LIN {X 0,Y 480.832,Z 518.896,A -85,B 0,C 180,E1 22694.82,E2 22694.82} C_VEL
LIN {X 0,Y 480.883,Z 518.889,A -85,B 0,C 180,E1 22691.393,E2 22691.393} C_VEL
LIN {X 0,Y 480.849,Z 518.879,A -85,B 0,C 180,E1 22687.888,E2 22687.888} C_VEL
LIN {X 0,Y 480.834,Z 518.897,A -85,B 0,C 180,E1 22684.413,E2 22684.413} C_VEL
LIN {X 0,Y 480.877,Z 518.875,A -85,B 0,C 180,E1 22680.953,E2 22680.953} C_VEL
LIN {X 0,Y 480.861,Z 518.895,A -85,B 0,C 180,E1 22677.498,E2 22677.498} C_VEL
LIN {X 0,Y 480.836,Z 518.893,A -85,B 0,C 180,E1 22674.032,E2 22674.032} C_VEL
LIN {X 0,Y 480.873,Z 518.893,A -85,B 0,C 180,E1 22670.546,E2 22670.546} C_VEL
LIN {X 0,Y 480.878,Z 518.894,A -85,B 0,C 180,E1 22667.023,E2 22667.023} C_VEL
LIN {X 0,Y 480.842,Z 518.893,A -85,B 0,C 180,E1 22663.573,E2 22663.573} C_VEL
LIN {X 0,Y 480.86,Z 518.889,A -85,B 0,C 180,E1 22660.017,E2 22660.017} C_VEL
LIN {X 0,Y 480.897,Z 518.897,A -85,B 0,C 180,E1 22656.47,E2 22656.47} C_VEL
LIN {X 0,Y 480.864,Z 518.888,A -85,B 0,C 180,E1 22652.859,E2 22652.859} C_VEL
LIN {X 0,Y 480.849,Z 518.893,A -85,B 0,C 180,E1 22649.373,E2 22649.373} C_VEL
LIN {X 0,Y 480.884,Z 518.892,A -85,B 0,C 180,E1 22645.841,E2 22645.841} C_VEL
LIN {X 0,Y 480.891,Z 518.896,A -85,B 0,C 180,E1 22642.19,E2 22642.19} C_VEL
LIN {X 0,Y 480.86,Z 518.9,A -85,B 0,C 180,E1 22638.642,E2 22638.642} C_VEL
LIN {X 0,Y 480.857,Z 518.892,A -85,B 0,C 180,E1 22634.986,E2 22634.986} C_VEL
LIN {X 0,Y 480.893,Z 518.896,A -85,B 0,C 180,E1 22631.387,E2 22631.387} C_VEL
LIN {X 0,Y 480.891,Z 518.896,A -85,B 0,C 180,E1 22627.806,E2 22627.806} C_VEL
LIN {X 0,Y 480.899,Z 519.178,A -85,B 0,C 180,E1 22626.666,E2 22626.666} C_VEL
LIN {X 0,Y 489.257,Z 542.949,A -85,B 0,C 180,E1 22623.815,E2 22623.815} C_VEL
LIN {X 0,Y 491.045,Z 549.01,A -85,B 0,C 180,E1 22623.147,E2 22623.147} C_VEL
LIN {X 0,Y 488.53,Z 593.414,A -85,B 0,C 180,E1 22619.418,E2 22619.418} C_VEL
LIN {X 0,Y 487.499,Z 615.888,A -85,B 0,C 180,E1 22617.597,E2 22617.597} C_VEL
LIN {X 0,Y 489.565,Z 633.074,A -85,B 0,C 180,E1 22617.228,E2 22617.228} C_VEL
LIN {X 0,Y 487.749,Z 821.161,A -85,B 0,C 180,E1 22614.405,E2 22614.405} C_VEL
LIN {X 0,Y 487.153,Z 840.046,A -85,B 0,C 180,E1 22613.909,E2 22613.909} C_VEL
LIN {X 0,Y 486.416,Z 858.284,A -85,B 0,C 180,E1 22613.213,E2 22613.213} C_VEL
LIN {X 0,Y 485.593,Z 875.737,A -85,B 0,C 180,E1 22612.327,E2 22612.327} C_VEL
LIN {X 0,Y 484.62,Z 892.847,A -85,B 0,C 180,E1 22611.228,E2 22611.228} C_VEL
LIN {X 0,Y 483.712,Z 909.068,A -85,B 0,C 180,E1 22609.941,E2 22609.941} C_VEL
LIN {X 0,Y 482.784,Z 924.925,A -85,B 0,C 180,E1 22608.411,E2 22608.411} C_VEL
LIN {X 0,Y 481.97,Z 939.095,A -85,B 0,C 180,E1 22606.76,E2 22606.76} C_VEL
LIN {X 0,Y 481.309,Z 951.749,A -85,B 0,C 180,E1 22604.989,E2 22604.989} C_VEL
LIN {X 0,Y 480.782,Z 962.938,A -85,B 0,C 180,E1 22603.102,E2 22603.102} C_VEL
LIN {X 0,Y 480.424,Z 972.395,A -85,B 0,C 180,E1 22601.161,E2 22601.161} C_VEL
LIN {X 0,Y 480.18,Z 980.439,A -85,B 0,C 180,E1 22599.106,E2 22599.106} C_VEL
LIN {X 0,Y 480.051,Z 986.651,A -85,B 0,C 180,E1 22597.06,E2 22597.06} C_VEL
LIN {X 0,Y 479.996,Z 991.41,A -85,B 0,C 180,E1 22594.9,E2 22594.9} C_VEL
LIN {X 0,Y 479.987,Z 994.401,A -85,B 0,C 180,E1 22592.747,E2 22592.747} C_VEL
LIN {X 0,Y 479.99,Z 995.698,A -85,B 0,C 180,E1 22590.598,E2 22590.598} C_VEL
LIN {X 0,Y 479.99,Z 995.327,A -85,B 0,C 180,E1 22588.45,E2 22588.45} C_VEL
LIN {X 0,Y 479.992,Z 993.281,A -85,B 0,C 180,E1 22586.299,E2 22586.299} C_VEL
LIN {X 0,Y 480.012,Z 989.511,A -85,B 0,C 180,E1 22584.144,E2 22584.144} C_VEL
LIN {X 0,Y 480.093,Z 984.297,A -85,B 0,C 180,E1 22582.102,E2 22582.102} C_VEL
LIN {X 0,Y 480.282,Z 976.985,A -85,B 0,C 180,E1 22579.964,E2 22579.964} C_VEL
LIN {X 0,Y 480.573,Z 968.08,A -85,B 0,C 180,E1 22577.921,E2 22577.921} C_VEL
LIN {X 0,Y 480.994,Z 958.057,A -85,B 0,C 180,E1 22576.049,E2 22576.049} C_VEL
LIN {X 0,Y 481.579,Z 946.227,A -85,B 0,C 180,E1 22574.221,E2 22574.221} C_VEL
LIN {X 0,Y 482.31,Z 932.666,A -85,B 0,C 180,E1 22572.479,E2 22572.479} C_VEL
LIN {X 0,Y 483.157,Z 918.064,A -85,B 0,C 180,E1 22570.918,E2 22570.918} C_VEL
LIN {X 0,Y 484.054,Z 902.156,A -85,B 0,C 180,E1 22569.509,E2 22569.509} C_VEL
LIN {X 0,Y 485.003,Z 885.243,A -85,B 0,C 180,E1 22568.285,E2 22568.285} C_VEL
LIN {X 0,Y 485.9,Z 867.99,A -85,B 0,C 180,E1 22567.284,E2 22567.284} C_VEL
LIN {X 0,Y 486.675,Z 850.244,A -85,B 0,C 180,E1 22566.483,E2 22566.483} C_VEL
LIN {X 0,Y 487.361,Z 831.618,A -85,B 0,C 180,E1 22565.872,E2 22565.872} C_VEL
LIN {X 0,Y 487.819,Z 812.718,A -85,B 0,C 180,E1 22565.472,E2 22565.472} C_VEL
LIN {X 0,Y 489.293,Z 630.035,A -85,B 0,C 180,E1 22562.747,E2 22562.747} C_VEL
LIN {X 0,Y 487.435,Z 615.346,A -85,B 0,C 180,E1 22562.393,E2 22562.393} C_VEL
LIN {X 0,Y 489.751,Z 570.848,A -85,B 0,C 180,E1 22558.701,E2 22558.701} C_VEL
LIN {X 0,Y 491.081,Z 548.213,A -85,B 0,C 180,E1 22556.751,E2 22556.751} C_VEL
LIN {X 0,Y 484.241,Z 528.175,A -85,B 0,C 180,E1 22554.341,E2 22554.341} C_VEL
LIN {X 0,Y 480.894,Z 519.106,A -85,B 0,C 180,E1 22553.106,E2 22553.106} C_VEL
LIN {X 0,Y 480.853,Z 518.898,A -85,B 0,C 180,E1 22549.556,E2 22549.556} C_VEL
LIN {X 0,Y 480.882,Z 518.9,A -85,B 0,C 180,E1 22546.006,E2 22546.006} C_VEL
LIN {X 0,Y 480.883,Z 518.896,A -85,B 0,C 180,E1 22542.436,E2 22542.436} C_VEL
LIN {X 0,Y 480.841,Z 518.893,A -85,B 0,C 180,E1 22538.959,E2 22538.959} C_VEL
LIN {X 0,Y 480.841,Z 518.896,A -85,B 0,C 180,E1 22535.315,E2 22535.315} C_VEL
LIN {X 0,Y 480.89,Z 518.889,A -85,B 0,C 180,E1 22531.878,E2 22531.878} C_VEL
LIN {X 0,Y 480.839,Z 518.896,A -85,B 0,C 180,E1 22528.436,E2 22528.436} C_VEL
LIN {X 0,Y 480.825,Z 518.897,A -85,B 0,C 180,E1 22524.838,E2 22524.838} C_VEL
LIN {X 0,Y 480.857,Z 518.901,A -85,B 0,C 180,E1 22521.339,E2 22521.339} C_VEL
LIN {X 0,Y 480.86,Z 518.894,A -85,B 0,C 180,E1 22517.784,E2 22517.784} C_VEL
LIN {X 0,Y 480.811,Z 518.889,A -85,B 0,C 180,E1 22514.315,E2 22514.315} C_VEL
LIN {X 0,Y 480.821,Z 518.897,A -85,B 0,C 180,E1 22510.787,E2 22510.787} C_VEL
LIN {X 0,Y 480.884,Z 518.899,A -85,B 0,C 180,E1 22507.286,E2 22507.286} C_VEL
LIN {X 0,Y 480.823,Z 518.892,A -85,B 0,C 180,E1 22503.815,E2 22503.815} C_VEL
LIN {X 0,Y 480.821,Z 518.891,A -85,B 0,C 180,E1 22500.238,E2 22500.238} C_VEL
LIN {X 0,Y 480.87,Z 518.896,A -85,B 0,C 180,E1 22496.781,E2 22496.781} C_VEL
LIN {X 0,Y 480.852,Z 518.898,A -85,B 0,C 180,E1 22493.313,E2 22493.313} C_VEL
LIN {X 0,Y 480.831,Z 518.894,A -85,B 0,C 180,E1 22489.819,E2 22489.819} C_VEL
LIN {X 0,Y 480.861,Z 518.89,A -85,B 0,C 180,E1 22486.288,E2 22486.288} C_VEL
LIN {X 0,Y 480.882,Z 518.891,A -85,B 0,C 180,E1 22482.827,E2 22482.827} C_VEL
LIN {X 0,Y 480.848,Z 518.897,A -85,B 0,C 180,E1 22479.299,E2 22479.299} C_VEL
LIN {X 0,Y 480.849,Z 518.892,A -85,B 0,C 180,E1 22475.596,E2 22475.596} C_VEL
LIN {X 0,Y 480.894,Z 518.897,A -85,B 0,C 180,E1 22472.073,E2 22472.073} C_VEL
LIN {X 0,Y 480.89,Z 518.895,A -85,B 0,C 180,E1 22468.47,E2 22468.47} C_VEL
LIN {X 0,Y 480.858,Z 518.902,A -85,B 0,C 180,E1 22464.977,E2 22464.977} C_VEL
LIN {X 0,Y 480.91,Z 519.174,A -85,B 0,C 180,E1 22462.637,E2 22462.637} C_VEL
LIN {X 0,Y 485.71,Z 535.44,A -85,B 0,C 180,E1 22459.884,E2 22459.884} C_VEL
LIN {X 0,Y 487.693,Z 543.443,A -85,B 0,C 180,E1 22458.614,E2 22458.614} C_VEL
LIN {X 0,Y 486.002,Z 570.518,A -85,B 0,C 180,E1 22455.042,E2 22455.042} C_VEL
LIN {X 0,Y 484.423,Z 600.385,A -85,B 0,C 180,E1 22451.173,E2 22451.173} C_VEL
LIN {X 0,Y 483.181,Z 628.631,A -85,B 0,C 180,E1 22447.575,E2 22447.575} C_VEL
LIN {X 0,Y 483.129,Z 631.811,A -85,B 0,C 180,E1 22447.207,E2 22447.207} C_VEL
LIN {X 0,Y 484.66,Z 640.368,A -85,B 0,C 180,E1 22446.962,E2 22446.962} C_VEL
LIN {X 0,Y 484.836,Z 645.811,A -85,B 0,C 180,E1 22446.867,E2 22446.867} C_VEL
LIN {X 0,Y 483.045,Z 654.53,A -85,B 0,C 180,E1 22446.817,E2 22446.817} C_VEL
LIN {X 0,Y 478.507,Z 669.749,A -85,B 0,C 180,E1 22446.799,E2 22446.799} C_VEL
LIN {X 0,Y 477.905,Z 675.336,A -85,B 0,C 180,E1 22446.738,E2 22446.738} C_VEL
LIN {X 0,Y 477.021,Z 749.526,A -85,B 0,C 180,E1 22445.515,E2 22445.515} C_VEL
LIN {X 0,Y 476.742,Z 763.894,A -85,B 0,C 180,E1 22445.07,E2 22445.07} C_VEL
LIN {X 0,Y 476.291,Z 778.064,A -85,B 0,C 180,E1 22444.41,E2 22444.41} C_VEL
LIN {X 0,Y 475.718,Z 791.572,A -85,B 0,C 180,E1 22443.552,E2 22443.552} C_VEL
LIN {X 0,Y 475.006,Z 804.939,A -85,B 0,C 180,E1 22442.426,E2 22442.426} C_VEL
LIN {X 0,Y 474.403,Z 815.997,A -85,B 0,C 180,E1 22441.225,E2 22441.225} C_VEL
LIN {X 0,Y 473.827,Z 826.024,A -85,B 0,C 180,E1 22439.855,E2 22439.855} C_VEL
LIN {X 0,Y 473.324,Z 834.493,A -85,B 0,C 180,E1 22438.374,E2 22438.374} C_VEL
LIN {X 0,Y 472.95,Z 841.657,A -85,B 0,C 180,E1 22436.759,E2 22436.759} C_VEL
LIN {X 0,Y 472.673,Z 847.643,A -85,B 0,C 180,E1 22434.891,E2 22434.891} C_VEL
LIN {X 0,Y 472.512,Z 851.491,A -85,B 0,C 180,E1 22433.042,E2 22433.042} C_VEL
LIN {X 0,Y 472.433,Z 853.501,A -85,B 0,C 180,E1 22431.214,E2 22431.214} C_VEL
LIN {X 0,Y 472.417,Z 853.747,A -85,B 0,C 180,E1 22429.273,E2 22429.273} C_VEL
LIN {X 0,Y 472.459,Z 852.063,A -85,B 0,C 180,E1 22427.358,E2 22427.358} C_VEL
LIN {X 0,Y 472.575,Z 848.779,A -85,B 0,C 180,E1 22425.584,E2 22425.584} C_VEL
LIN {X 0,Y 472.778,Z 843.721,A -85,B 0,C 180,E1 22423.824,E2 22423.824} C_VEL
LIN {X 0,Y 473.073,Z 837.213,A -85,B 0,C 180,E1 22422.199,E2 22422.199} C_VEL
LIN {X 0,Y 473.491,Z 829.444,A -85,B 0,C 180,E1 22420.707,E2 22420.707} C_VEL
LIN {X 0,Y 474.044,Z 819.355,A -85,B 0,C 180,E1 22419.207,E2 22419.207} C_VEL
LIN {X 0,Y 474.639,Z 808.412,A -85,B 0,C 180,E1 22417.929,E2 22417.929} C_VEL
LIN {X 0,Y 475.291,Z 795.658,A -85,B 0,C 180,E1 22416.763,E2 22416.763} C_VEL
LIN {X 0,Y 475.916,Z 781.501,A -85,B 0,C 180,E1 22415.786,E2 22415.786} C_VEL
LIN {X 0,Y 476.386,Z 767.869,A -85,B 0,C 180,E1 22415.092,E2 22415.092} C_VEL
LIN {X 0,Y 476.752,Z 752.577,A -85,B 0,C 180,E1 22414.558,E2 22414.558} C_VEL
LIN {X 0,Y 476.981,Z 731.635,A -85,B 0,C 180,E1 22414.162,E2 22414.162} C_VEL
LIN {X 0,Y 477.695,Z 645.512,A -85,B 0,C 180,E1 22412.808,E2 22412.808} C_VEL
LIN {X 0,Y 475.264,Z 632.071,A -85,B 0,C 180,E1 22412.47,E2 22412.47} C_VEL
LIN {X 0,Y 475.368,Z 627.356,A -85,B 0,C 180,E1 22411.927,E2 22411.927} C_VEL
LIN {X 0,Y 476.674,Z 598.333,A -85,B 0,C 180,E1 22408.196,E2 22408.196} C_VEL
LIN {X 0,Y 478.235,Z 569.754,A -85,B 0,C 180,E1 22404.48,E2 22404.48} C_VEL
LIN {X 0,Y 479.675,Z 544.41,A -85,B 0,C 180,E1 22401.126,E2 22401.126} C_VEL
LIN {X 0,Y 474.789,Z 526.621,A -85,B 0,C 180,E1 22398.308,E2 22398.308} C_VEL
LIN {X 0,Y 472.922,Z 519.987,A -85,B 0,C 180,E1 22397.174,E2 22397.174} C_VEL
LIN {X 0,Y 472.912,Z 519.892,A -85,B 0,C 180,E1 22393.716,E2 22393.716} C_VEL
LIN {X 0,Y 472.875,Z 519.888,A -85,B 0,C 180,E1 22390.208,E2 22390.208} C_VEL
LIN {X 0,Y 472.888,Z 519.86,A -85,B 0,C 180,E1 22386.71,E2 22386.71} C_VEL
LIN {X 0,Y 472.93,Z 519.89,A -85,B 0,C 180,E1 22383.15,E2 22383.15} C_VEL
LIN {X 0,Y 472.867,Z 519.859,A -85,B 0,C 180,E1 22379.786,E2 22379.786} C_VEL
LIN {X 0,Y 472.872,Z 519.89,A -85,B 0,C 180,E1 22376.069,E2 22376.069} C_VEL
LIN {X 0,Y 472.923,Z 519.88,A -85,B 0,C 180,E1 22372.645,E2 22372.645} C_VEL
LIN {X 0,Y 472.889,Z 519.891,A -85,B 0,C 180,E1 22369.196,E2 22369.196} C_VEL
LIN {X 0,Y 472.875,Z 519.888,A -85,B 0,C 180,E1 22365.586,E2 22365.586} C_VEL
LIN {X 0,Y 472.905,Z 519.876,A -85,B 0,C 180,E1 22362.085,E2 22362.085} C_VEL
LIN {X 0,Y 472.921,Z 519.886,A -85,B 0,C 180,E1 22358.587,E2 22358.587} C_VEL
LIN {X 0,Y 472.88,Z 519.881,A -85,B 0,C 180,E1 22355.092,E2 22355.092} C_VEL
LIN {X 0,Y 472.893,Z 519.887,A -85,B 0,C 180,E1 22351.483,E2 22351.483} C_VEL
LIN {X 0,Y 472.942,Z 519.879,A -85,B 0,C 180,E1 22348.129,E2 22348.129} C_VEL
LIN {X 0,Y 472.891,Z 519.876,A -85,B 0,C 180,E1 22344.616,E2 22344.616} C_VEL
LIN {X 0,Y 472.891,Z 519.887,A -85,B 0,C 180,E1 22341.066,E2 22341.066} C_VEL
LIN {X 0,Y 472.938,Z 519.865,A -85,B 0,C 180,E1 22337.556,E2 22337.556} C_VEL
LIN {X 0,Y 472.912,Z 519.886,A -85,B 0,C 180,E1 22334.072,E2 22334.072} C_VEL
LIN {X 0,Y 472.89,Z 519.879,A -85,B 0,C 180,E1 22330.477,E2 22330.477} C_VEL
LIN {X 0,Y 472.915,Z 519.88,A -85,B 0,C 180,E1 22326.922,E2 22326.922} C_VEL
LIN {X 0,Y 472.945,Z 519.883,A -85,B 0,C 180,E1 22323.394,E2 22323.394} C_VEL
LIN {X 0,Y 472.899,Z 519.866,A -85,B 0,C 180,E1 22319.879,E2 22319.879} C_VEL
LIN {X 0,Y 472.901,Z 519.887,A -85,B 0,C 180,E1 22316.242,E2 22316.242} C_VEL
LIN {X 0,Y 472.942,Z 519.866,A -85,B 0,C 180,E1 22312.713,E2 22312.713} C_VEL
LIN {X 0,Y 472.934,Z 519.887,A -85,B 0,C 180,E1 22309.155,E2 22309.155} C_VEL
LIN {X 0,Y 472.902,Z 519.877,A -85,B 0,C 180,E1 22305.678,E2 22305.678} C_VEL
LIN {X 0,Y 472.92,Z 519.885,A -85,B 0,C 180,E1 22302.053,E2 22302.053} C_VEL
LIN {X 0,Y 472.957,Z 519.874,A -85,B 0,C 180,E1 22298.417,E2 22298.417} C_VEL
LIN {X 0,Y 472.933,Z 519.885,A -85,B 0,C 180,E1 22294.798,E2 22294.798} C_VEL
LIN {X 0,Y 472.908,Z 519.887,A -85,B 0,C 180,E1 22291.319,E2 22291.319} C_VEL
LIN {X 0,Y 472.94,Z 519.883,A -85,B 0,C 180,E1 22287.808,E2 22287.808} C_VEL
LIN {X 0,Y 472.954,Z 519.88,A -85,B 0,C 180,E1 22284.155,E2 22284.155} C_VEL
LIN {X 0,Y 472.92,Z 519.882,A -85,B 0,C 180,E1 22280.634,E2 22280.634} C_VEL
LIN {X 0,Y 472.916,Z 519.886,A -85,B 0,C 180,E1 22277.011,E2 22277.011} C_VEL
LIN {X 0,Y 472.944,Z 519.884,A -85,B 0,C 180,E1 22273.397,E2 22273.397} C_VEL
LIN {X 0,Y 472.953,Z 519.884,A -85,B 0,C 180,E1 22269.832,E2 22269.832} C_VEL
LIN {X 0,Y 472.984,Z 520.157,A -85,B 0,C 180,E1 22267.197,E2 22267.197} C_VEL
LIN {X 0,Y 481.63,Z 544.659,A -85,B 0,C 180,E1 22264.19,E2 22264.19} C_VEL
LIN {X 0,Y 483.726,Z 551.404,A -85,B 0,C 180,E1 22263.424,E2 22263.424} C_VEL
LIN {X 0,Y 481.019,Z 595.587,A -85,B 0,C 180,E1 22259.65,E2 22259.65} C_VEL
LIN {X 0,Y 479.984,Z 615.915,A -85,B 0,C 180,E1 22257.965,E2 22257.965} C_VEL
LIN {X 0,Y 482.128,Z 634.091,A -85,B 0,C 180,E1 22257.565,E2 22257.565} C_VEL
LIN {X 0,Y 480.215,Z 820.44,A -85,B 0,C 180,E1 22254.735,E2 22254.735} C_VEL
LIN {X 0,Y 479.585,Z 839.412,A -85,B 0,C 180,E1 22254.231,E2 22254.231} C_VEL
LIN {X 0,Y 478.821,Z 857.057,A -85,B 0,C 180,E1 22253.551,E2 22253.551} C_VEL
LIN {X 0,Y 477.92,Z 874.81,A -85,B 0,C 180,E1 22252.64,E2 22252.64} C_VEL
LIN {X 0,Y 476.888,Z 891.93,A -85,B 0,C 180,E1 22251.525,E2 22251.525} C_VEL
LIN {X 0,Y 475.918,Z 908.149,A -85,B 0,C 180,E1 22250.218,E2 22250.218} C_VEL
LIN {X 0,Y 474.929,Z 923.994,A -85,B 0,C 180,E1 22248.663,E2 22248.663} C_VEL
LIN {X 0,Y 474.09,Z 937.665,A -85,B 0,C 180,E1 22247.047,E2 22247.047} C_VEL
LIN {X 0,Y 473.365,Z 950.783,A -85,B 0,C 180,E1 22245.184,E2 22245.184} C_VEL
LIN {X 0,Y 472.836,Z 961.624,A -85,B 0,C 180,E1 22243.326,E2 22243.326} C_VEL
LIN {X 0,Y 472.465,Z 971.123,A -85,B 0,C 180,E1 22241.351,E2 22241.351} C_VEL
LIN {X 0,Y 472.229,Z 979.203,A -85,B 0,C 180,E1 22239.261,E2 22239.261} C_VEL
LIN {X 0,Y 472.101,Z 985.44,A -85,B 0,C 180,E1 22237.179,E2 22237.179} C_VEL
LIN {X 0,Y 472.063,Z 990.218,A -85,B 0,C 180,E1 22234.983,E2 22234.983} C_VEL
LIN {X 0,Y 472.067,Z 993.22,A -85,B 0,C 180,E1 22232.794,E2 22232.794} C_VEL
LIN {X 0,Y 472.077,Z 994.52,A -85,B 0,C 180,E1 22230.608,E2 22230.608} C_VEL
LIN {X 0,Y 472.075,Z 994.144,A -85,B 0,C 180,E1 22228.424,E2 22228.424} C_VEL
LIN {X 0,Y 472.069,Z 992.083,A -85,B 0,C 180,E1 22226.237,E2 22226.237} C_VEL
LIN {X 0,Y 472.075,Z 988.291,A -85,B 0,C 180,E1 22224.045,E2 22224.045} C_VEL
LIN {X 0,Y 472.14,Z 983.045,A -85,B 0,C 180,E1 22221.968,E2 22221.968} C_VEL
LIN {X 0,Y 472.318,Z 975.94,A -85,B 0,C 180,E1 22219.855,E2 22219.855} C_VEL
LIN {X 0,Y 472.606,Z 967.105,A -85,B 0,C 180,E1 22217.789,E2 22217.789} C_VEL
LIN {X 0,Y 473.061,Z 956.667,A -85,B 0,C 180,E1 22215.811,E2 22215.811} C_VEL
LIN {X 0,Y 473.671,Z 944.769,A -85,B 0,C 180,E1 22213.95,E2 22213.95} C_VEL
LIN {X 0,Y 474.438,Z 931.388,A -85,B 0,C 180,E1 22212.21,E2 22212.21} C_VEL
LIN {X 0,Y 475.356,Z 916.422,A -85,B 0,C 180,E1 22210.593,E2 22210.593} C_VEL
LIN {X 0,Y 476.317,Z 900.378,A -85,B 0,C 180,E1 22209.161,E2 22209.161} C_VEL
LIN {X 0,Y 477.293,Z 884.216,A -85,B 0,C 180,E1 22207.981,E2 22207.981} C_VEL
LIN {X 0,Y 478.223,Z 867.38,A -85,B 0,C 180,E1 22206.988,E2 22206.988} C_VEL
LIN {X 0,Y 479.075,Z 849.388,A -85,B 0,C 180,E1 22206.163,E2 22206.163} C_VEL
LIN {X 0,Y 479.808,Z 830.665,A -85,B 0,C 180,E1 22205.541,E2 22205.541} C_VEL
LIN {X 0,Y 480.296,Z 811.558,A -85,B 0,C 180,E1 22205.135,E2 22205.135} C_VEL
LIN {X 0,Y 481.901,Z 631.165,A -85,B 0,C 180,E1 22202.404,E2 22202.404} C_VEL
LIN {X 0,Y 479.957,Z 615.552,A -85,B 0,C 180,E1 22202.022,E2 22202.022} C_VEL
LIN {X 0,Y 482.471,Z 571.77,A -85,B 0,C 180,E1 22198.313,E2 22198.313} C_VEL
LIN {X 0,Y 483.89,Z 551.303,A -85,B 0,C 180,E1 22196.521,E2 22196.521} C_VEL
LIN {X 0,Y 477.58,Z 532.578,A -85,B 0,C 180,E1 22194.22,E2 22194.22} C_VEL
LIN {X 0,Y 472.984,Z 520.089,A -85,B 0,C 180,E1 22192.493,E2 22192.493} C_VEL
LIN {X 0,Y 472.921,Z 519.884,A -85,B 0,C 180,E1 22189.006,E2 22189.006} C_VEL
LIN {X 0,Y 472.91,Z 519.89,A -85,B 0,C 180,E1 22185.424,E2 22185.424} C_VEL
LIN {X 0,Y 472.942,Z 519.881,A -85,B 0,C 180,E1 22181.918,E2 22181.918} C_VEL
LIN {X 0,Y 472.94,Z 519.878,A -85,B 0,C 180,E1 22178.349,E2 22178.349} C_VEL
LIN {X 0,Y 472.898,Z 519.885,A -85,B 0,C 180,E1 22174.811,E2 22174.811} C_VEL
LIN {X 0,Y 472.896,Z 519.888,A -85,B 0,C 180,E1 22171.107,E2 22171.107} C_VEL
LIN {X 0,Y 472.94,Z 519.878,A -85,B 0,C 180,E1 22167.66,E2 22167.66} C_VEL
LIN {X 0,Y 472.913,Z 519.881,A -85,B 0,C 180,E1 22164.082,E2 22164.082} C_VEL
LIN {X 0,Y 472.88,Z 519.889,A -85,B 0,C 180,E1 22160.677,E2 22160.677} C_VEL
LIN {X 0,Y 472.905,Z 519.891,A -85,B 0,C 180,E1 22157.147,E2 22157.147} C_VEL
LIN {X 0,Y 472.911,Z 519.877,A -85,B 0,C 180,E1 22153.697,E2 22153.697} C_VEL
LIN {X 0,Y 472.869,Z 519.885,A -85,B 0,C 180,E1 22150.231,E2 22150.231} C_VEL
LIN {X 0,Y 472.88,Z 519.89,A -85,B 0,C 180,E1 22146.556,E2 22146.556} C_VEL
LIN {X 0,Y 472.93,Z 519.886,A -85,B 0,C 180,E1 22143.03,E2 22143.03} C_VEL
LIN {X 0,Y 472.902,Z 519.878,A -85,B 0,C 180,E1 22139.515,E2 22139.515} C_VEL
LIN {X 0,Y 472.885,Z 519.886,A -85,B 0,C 180,E1 22135.999,E2 22135.999} C_VEL
LIN {X 0,Y 472.917,Z 519.887,A -85,B 0,C 180,E1 22132.468,E2 22132.468} C_VEL
LIN {X 0,Y 472.945,Z 519.886,A -85,B 0,C 180,E1 22128.908,E2 22128.908} C_VEL
LIN {X 0,Y 472.902,Z 519.883,A -85,B 0,C 180,E1 22125.427,E2 22125.427} C_VEL
LIN {X 0,Y 472.905,Z 519.885,A -85,B 0,C 180,E1 22121.765,E2 22121.765} C_VEL
LIN {X 0,Y 472.954,Z 519.882,A -85,B 0,C 180,E1 22118.286,E2 22118.286} C_VEL
LIN {X 0,Y 472.94,Z 519.885,A -85,B 0,C 180,E1 22114.719,E2 22114.719} C_VEL
LIN {X 0,Y 472.914,Z 519.89,A -85,B 0,C 180,E1 22111.18,E2 22111.18} C_VEL
LIN {X 0,Y 472.924,Z 519.887,A -85,B 0,C 180,E1 22107.508,E2 22107.508} C_VEL
LIN {X 0,Y 472.953,Z 519.882,A -85,B 0,C 180,E1 22104.005,E2 22104.005} C_VEL
LIN {X 0,Y 472.97,Z 520.223,A -85,B 0,C 180,E1 22103.203,E2 22103.203} C_VEL
LIN {X 0,Y 477.948,Z 536.611,A -85,B 0,C 180,E1 22100.353,E2 22100.353} C_VEL
LIN {X 0,Y 480.275,Z 546.322,A -85,B 0,C 180,E1 22098.783,E2 22098.783} C_VEL
LIN {X 0,Y 478.464,Z 573.198,A -85,B 0,C 180,E1 22095.184,E2 22095.184} C_VEL
LIN {X 0,Y 476.803,Z 602.516,A -85,B 0,C 180,E1 22091.336,E2 22091.336} C_VEL
LIN {X 0,Y 475.472,Z 631.275,A -85,B 0,C 180,E1 22087.634,E2 22087.634} C_VEL
LIN {X 0,Y 476.252,Z 635.903,A -85,B 0,C 180,E1 22087.465,E2 22087.465} C_VEL
LIN {X 0,Y 478.239,Z 648.3,A -85,B 0,C 180,E1 22087.16,E2 22087.16} C_VEL
LIN {X 0,Y 477.905,Z 675.336,A -85,B 0,C 180,E1 22086.738,E2 22086.738} C_VEL
LIN {X 0,Y 476.914,Z 683.01,A -85,B 0,C 180,E1 22086.662,E2 22086.662} C_VEL
LIN {X 0,Y 470.854,Z 703.38,A -85,B 0,C 180,E1 22086.627,E2 22086.627} C_VEL
LIN {X 0,Y 470.071,Z 709.967,A -85,B 0,C 180,E1 22086.554,E2 22086.554} C_VEL
LIN {X 0,Y 469.547,Z 750.832,A -85,B 0,C 180,E1 22085.839,E2 22085.839} C_VEL
LIN {X 0,Y 469.223,Z 766.124,A -85,B 0,C 180,E1 22085.342,E2 22085.342} C_VEL
LIN {X 0,Y 468.664,Z 781.639,A -85,B 0,C 180,E1 22084.57,E2 22084.57} C_VEL
LIN {X 0,Y 468.019,Z 794.839,A -85,B 0,C 180,E1 22083.666,E2 22083.666} C_VEL
LIN {X 0,Y 467.342,Z 806.736,A -85,B 0,C 180,E1 22082.62,E2 22082.62} C_VEL
LIN {X 0,Y 466.641,Z 818.407,A -85,B 0,C 180,E1 22081.3,E2 22081.3} C_VEL
LIN {X 0,Y 466.024,Z 828.108,A -85,B 0,C 180,E1 22079.912,E2 22079.912} C_VEL
LIN {X 0,Y 465.457,Z 837.066,A -85,B 0,C 180,E1 22078.268,E2 22078.268} C_VEL
LIN {X 0,Y 465.042,Z 844.063,A -85,B 0,C 180,E1 22076.561,E2 22076.561} C_VEL
LIN {X 0,Y 464.774,Z 849.342,A -85,B 0,C 180,E1 22074.791,E2 22074.791} C_VEL
LIN {X 0,Y 464.606,Z 852.992,A -85,B 0,C 180,E1 22072.914,E2 22072.914} C_VEL
LIN {X 0,Y 464.519,Z 854.777,A -85,B 0,C 180,E1 22071.064,E2 22071.064} C_VEL
LIN {X 0,Y 464.505,Z 854.911,A -85,B 0,C 180,E1 22069.225,E2 22069.225} C_VEL
LIN {X 0,Y 464.555,Z 853.186,A -85,B 0,C 180,E1 22067.275,E2 22067.275} C_VEL
LIN {X 0,Y 464.69,Z 849.763,A -85,B 0,C 180,E1 22065.43,E2 22065.43} C_VEL
LIN {X 0,Y 464.933,Z 844.427,A -85,B 0,C 180,E1 22063.578,E2 22063.578} C_VEL
LIN {X 0,Y 465.316,Z 837.086,A -85,B 0,C 180,E1 22061.776,E2 22061.776} C_VEL
LIN {X 0,Y 465.791,Z 828.933,A -85,B 0,C 180,E1 22060.261,E2 22060.261} C_VEL
LIN {X 0,Y 466.405,Z 818.806,A -85,B 0,C 180,E1 22058.781,E2 22058.781} C_VEL
LIN {X 0,Y 467.082,Z 806.99,A -85,B 0,C 180,E1 22057.439,E2 22057.439} C_VEL
LIN {X 0,Y 467.725,Z 795.077,A -85,B 0,C 180,E1 22056.38,E2 22056.38} C_VEL
LIN {X 0,Y 468.36,Z 781.557,A -85,B 0,C 180,E1 22055.449,E2 22055.449} C_VEL
LIN {X 0,Y 468.888,Z 766.723,A -85,B 0,C 180,E1 22054.707,E2 22054.707} C_VEL
LIN {X 0,Y 469.233,Z 751.884,A -85,B 0,C 180,E1 22054.207,E2 22054.207} C_VEL
LIN {X 0,Y 469.498,Z 728.892,A -85,B 0,C 180,E1 22053.784,E2 22053.784} C_VEL
LIN {X 0,Y 470.238,Z 646.544,A -85,B 0,C 180,E1 22052.465,E2 22052.465} C_VEL
LIN {X 0,Y 467.584,Z 631.78,A -85,B 0,C 180,E1 22052.082,E2 22052.082} C_VEL
LIN {X 0,Y 468.299,Z 614.44,A -85,B 0,C 180,E1 22049.876,E2 22049.876} C_VEL
LIN {X 0,Y 469.841,Z 585.517,A -85,B 0,C 180,E1 22046.094,E2 22046.094} C_VEL
LIN {X 0,Y 471.577,Z 557.087,A -85,B 0,C 180,E1 22042.323,E2 22042.323} C_VEL
LIN {X 0,Y 472.045,Z 546.316,A -85,B 0,C 180,E1 22040.859,E2 22040.859} C_VEL
LIN {X 0,Y 467.151,Z 528.61,A -85,B 0,C 180,E1 22037.998,E2 22037.998} C_VEL
LIN {X 0,Y 464.958,Z 521.007,A -85,B 0,C 180,E1 22036.697,E2 22036.697} C_VEL
LIN {X 0,Y 464.988,Z 520.876,A -85,B 0,C 180,E1 22033.253,E2 22033.253} C_VEL
LIN {X 0,Y 464.966,Z 520.876,A -85,B 0,C 180,E1 22029.649,E2 22029.649} C_VEL
LIN {X 0,Y 464.93,Z 520.849,A -85,B 0,C 180,E1 22026.153,E2 22026.153} C_VEL
LIN {X 0,Y 464.951,Z 520.878,A -85,B 0,C 180,E1 22022.601,E2 22022.601} C_VEL
LIN {X 0,Y 464.984,Z 520.839,A -85,B 0,C 180,E1 22019.076,E2 22019.076} C_VEL
LIN {X 0,Y 464.938,Z 520.879,A -85,B 0,C 180,E1 22015.559,E2 22015.559} C_VEL
LIN {X 0,Y 464.934,Z 520.875,A -85,B 0,C 180,E1 22011.89,E2 22011.89} C_VEL
LIN {X 0,Y 464.981,Z 520.867,A -85,B 0,C 180,E1 22008.445,E2 22008.445} C_VEL
LIN {X 0,Y 464.97,Z 520.877,A -85,B 0,C 180,E1 22004.856,E2 22004.856} C_VEL
LIN {X 0,Y 464.937,Z 520.865,A -85,B 0,C 180,E1 22001.317,E2 22001.317} C_VEL
LIN {X 0,Y 464.948,Z 520.878,A -85,B 0,C 180,E1 21997.643,E2 21997.643} C_VEL
LIN {X 0,Y 464.994,Z 520.858,A -85,B 0,C 180,E1 21994.126,E2 21994.126} C_VEL
LIN {X 0,Y 464.97,Z 520.878,A -85,B 0,C 180,E1 21990.497,E2 21990.497} C_VEL
LIN {X 0,Y 464.944,Z 520.865,A -85,B 0,C 180,E1 21986.985,E2 21986.985} C_VEL
LIN {X 0,Y 464.971,Z 520.875,A -85,B 0,C 180,E1 21983.442,E2 21983.442} C_VEL
LIN {X 0,Y 464.991,Z 520.871,A -85,B 0,C 180,E1 21979.993,E2 21979.993} C_VEL
LIN {X 0,Y 464.951,Z 520.86,A -85,B 0,C 180,E1 21976.454,E2 21976.454} C_VEL
LIN {X 0,Y 464.956,Z 520.876,A -85,B 0,C 180,E1 21972.797,E2 21972.797} C_VEL
LIN {X 0,Y 464.998,Z 520.85,A -85,B 0,C 180,E1 21969.281,E2 21969.281} C_VEL
LIN {X 0,Y 464.975,Z 520.872,A -85,B 0,C 180,E1 21965.801,E2 21965.801} C_VEL
LIN {X 0,Y 464.956,Z 520.869,A -85,B 0,C 180,E1 21962.219,E2 21962.219} C_VEL
LIN {X 0,Y 464.979,Z 520.869,A -85,B 0,C 180,E1 21958.645,E2 21958.645} C_VEL
LIN {X 0,Y 465.01,Z 520.871,A -85,B 0,C 180,E1 21955.066,E2 21955.066} C_VEL
LIN {X 0,Y 464.969,Z 520.859,A -85,B 0,C 180,E1 21951.538,E2 21951.538} C_VEL
LIN {X 0,Y 464.965,Z 520.875,A -85,B 0,C 180,E1 21947.961,E2 21947.961} C_VEL
LIN {X 0,Y 465.001,Z 520.865,A -85,B 0,C 180,E1 21944.409,E2 21944.409} C_VEL
LIN {X 0,Y 465.007,Z 520.872,A -85,B 0,C 180,E1 21940.793,E2 21940.793} C_VEL
LIN {X 0,Y 464.969,Z 520.872,A -85,B 0,C 180,E1 21937.228,E2 21937.228} C_VEL
LIN {X 0,Y 464.973,Z 520.863,A -85,B 0,C 180,E1 21933.569,E2 21933.569} C_VEL
LIN {X 0,Y 465.019,Z 520.868,A -85,B 0,C 180,E1 21930.05,E2 21930.05} C_VEL
LIN {X 0,Y 465.003,Z 520.878,A -85,B 0,C 180,E1 21926.454,E2 21926.454} C_VEL
LIN {X 0,Y 464.977,Z 520.877,A -85,B 0,C 180,E1 21922.826,E2 21922.826} C_VEL
LIN {X 0,Y 464.981,Z 520.876,A -85,B 0,C 180,E1 21919.179,E2 21919.179} C_VEL
LIN {X 0,Y 465.01,Z 520.868,A -85,B 0,C 180,E1 21915.547,E2 21915.547} C_VEL
LIN {X 0,Y 465.012,Z 520.873,A -85,B 0,C 180,E1 21911.93,E2 21911.93} C_VEL
LIN {X 0,Y 464.986,Z 520.873,A -85,B 0,C 180,E1 21908.292,E2 21908.292} C_VEL
LIN {X 0,Y 465.082,Z 521.307,A -85,B 0,C 180,E1 21907.715,E2 21907.715} C_VEL
LIN {X 0,Y 473.934,Z 546.291,A -85,B 0,C 180,E1 21904.575,E2 21904.575} C_VEL
LIN {X 0,Y 476.336,Z 554.301,A -85,B 0,C 180,E1 21903.651,E2 21903.651} C_VEL
LIN {X 0,Y 473.415,Z 599.238,A -85,B 0,C 180,E1 21899.756,E2 21899.756} C_VEL
LIN {X 0,Y 472.526,Z 616.422,A -85,B 0,C 180,E1 21898.328,E2 21898.328} C_VEL
LIN {X 0,Y 474.712,Z 634.985,A -85,B 0,C 180,E1 21897.915,E2 21897.915} C_VEL
LIN {X 0,Y 472.676,Z 819.885,A -85,B 0,C 180,E1 21895.065,E2 21895.065} C_VEL
LIN {X 0,Y 472.015,Z 838.798,A -85,B 0,C 180,E1 21894.556,E2 21894.556} C_VEL
LIN {X 0,Y 471.184,Z 856.725,A -85,B 0,C 180,E1 21893.853,E2 21893.853} C_VEL
LIN {X 0,Y 470.243,Z 874.144,A -85,B 0,C 180,E1 21892.945,E2 21892.945} C_VEL
LIN {X 0,Y 469.175,Z 891.01,A -85,B 0,C 180,E1 21891.831,E2 21891.831} C_VEL
LIN {X 0,Y 468.134,Z 907.23,A -85,B 0,C 180,E1 21890.504,E2 21890.504} C_VEL
LIN {X 0,Y 467.124,Z 922.488,A -85,B 0,C 180,E1 21888.987,E2 21888.987} C_VEL
LIN {X 0,Y 466.224,Z 936.238,A -85,B 0,C 180,E1 21887.343,E2 21887.343} C_VEL
LIN {X 0,Y 465.447,Z 949.417,A -85,B 0,C 180,E1 21885.449,E2 21885.449} C_VEL
LIN {X 0,Y 464.888,Z 960.318,A -85,B 0,C 180,E1 21883.557,E2 21883.557} C_VEL
LIN {X 0,Y 464.502,Z 969.85,A -85,B 0,C 180,E1 21881.548,E2 21881.548} C_VEL
LIN {X 0,Y 464.271,Z 977.964,A -85,B 0,C 180,E1 21879.421,E2 21879.421} C_VEL
LIN {X 0,Y 464.147,Z 984.549,A -85,B 0,C 180,E1 21877.178,E2 21877.178} C_VEL
LIN {X 0,Y 464.128,Z 989.245,A -85,B 0,C 180,E1 21874.944,E2 21874.944} C_VEL
LIN {X 0,Y 464.146,Z 992.16,A -85,B 0,C 180,E1 21872.718,E2 21872.718} C_VEL
LIN {X 0,Y 464.161,Z 993.365,A -85,B 0,C 180,E1 21870.495,E2 21870.495} C_VEL
LIN {X 0,Y 464.162,Z 992.846,A -85,B 0,C 180,E1 21868.205,E2 21868.205} C_VEL
LIN {X 0,Y 464.147,Z 990.542,A -85,B 0,C 180,E1 21865.925,E2 21865.925} C_VEL
LIN {X 0,Y 464.147,Z 986.527,A -85,B 0,C 180,E1 21863.695,E2 21863.695} C_VEL
LIN {X 0,Y 464.219,Z 980.667,A -85,B 0,C 180,E1 21861.456,E2 21861.456} C_VEL
LIN {X 0,Y 464.399,Z 973.299,A -85,B 0,C 180,E1 21859.332,E2 21859.332} C_VEL
LIN {X 0,Y 464.72,Z 963.947,A -85,B 0,C 180,E1 21857.199,E2 21857.199} C_VEL
LIN {X 0,Y 465.241,Z 953.058,A -85,B 0,C 180,E1 21855.185,E2 21855.185} C_VEL
LIN {X 0,Y 465.928,Z 940.645,A -85,B 0,C 180,E1 21853.291,E2 21853.291} C_VEL
LIN {X 0,Y 466.804,Z 926.664,A -85,B 0,C 180,E1 21851.521,E2 21851.521} C_VEL
LIN {X 0,Y 467.794,Z 911.6,A -85,B 0,C 180,E1 21849.941,E2 21849.941} C_VEL
LIN {X 0,Y 468.816,Z 895.508,A -85,B 0,C 180,E1 21848.549,E2 21848.549} C_VEL
LIN {X 0,Y 469.921,Z 878.426,A -85,B 0,C 180,E1 21847.353,E2 21847.353} C_VEL
LIN {X 0,Y 470.886,Z 860.898,A -85,B 0,C 180,E1 21846.377,E2 21846.377} C_VEL
LIN {X 0,Y 471.766,Z 842.527,A -85,B 0,C 180,E1 21845.601,E2 21845.601} C_VEL
LIN {X 0,Y 472.501,Z 823.565,A -85,B 0,C 180,E1 21845.043,E2 21845.043} C_VEL
LIN {X 0,Y 472.923,Z 797.591,A -85,B 0,C 180,E1 21844.59,E2 21844.59} C_VEL
LIN {X 0,Y 474.499,Z 632.1,A -85,B 0,C 180,E1 21842.045,E2 21842.045} C_VEL
LIN {X 0,Y 472.496,Z 615.782,A -85,B 0,C 180,E1 21841.641,E2 21841.641} C_VEL
LIN {X 0,Y 475.269,Z 571.955,A -85,B 0,C 180,E1 21837.847,E2 21837.847} C_VEL
LIN {X 0,Y 476.504,Z 553.622,A -85,B 0,C 180,E1 21836.195,E2 21836.195} C_VEL
LIN {X 0,Y 469.981,Z 534.337,A -85,B 0,C 180,E1 21833.747,E2 21833.747} C_VEL
LIN {X 0,Y 465.019,Z 521.112,A -85,B 0,C 180,E1 21831.856,E2 21831.856} C_VEL
LIN {X 0,Y 465.021,Z 520.872,A -85,B 0,C 180,E1 21828.439,E2 21828.439} C_VEL
LIN {X 0,Y 464.985,Z 520.874,A -85,B 0,C 180,E1 21824.805,E2 21824.805} C_VEL
LIN {X 0,Y 464.965,Z 520.877,A -85,B 0,C 180,E1 21821.149,E2 21821.149} C_VEL
LIN {X 0,Y 464.974,Z 520.88,A -85,B 0,C 180,E1 21817.485,E2 21817.485} C_VEL
LIN {X 0,Y 465.007,Z 520.877,A -85,B 0,C 180,E1 21813.842,E2 21813.842} C_VEL
LIN {X 0,Y 464.988,Z 520.875,A -85,B 0,C 180,E1 21810.195,E2 21810.195} C_VEL
LIN {X 0,Y 464.949,Z 520.877,A -85,B 0,C 180,E1 21806.708,E2 21806.708} C_VEL
LIN {X 0,Y 464.954,Z 520.874,A -85,B 0,C 180,E1 21803.032,E2 21803.032} C_VEL
LIN {X 0,Y 464.997,Z 520.865,A -85,B 0,C 180,E1 21799.599,E2 21799.599} C_VEL
LIN {X 0,Y 464.956,Z 520.88,A -85,B 0,C 180,E1 21795.977,E2 21795.977} C_VEL
LIN {X 0,Y 464.933,Z 520.88,A -85,B 0,C 180,E1 21792.419,E2 21792.419} C_VEL
LIN {X 0,Y 464.949,Z 520.874,A -85,B 0,C 180,E1 21788.782,E2 21788.782} C_VEL
LIN {X 0,Y 464.991,Z 520.866,A -85,B 0,C 180,E1 21785.305,E2 21785.305} C_VEL
LIN {X 0,Y 464.952,Z 520.88,A -85,B 0,C 180,E1 21781.725,E2 21781.725} C_VEL
LIN {X 0,Y 464.946,Z 520.878,A -85,B 0,C 180,E1 21778.151,E2 21778.151} C_VEL
LIN {X 0,Y 464.978,Z 520.869,A -85,B 0,C 180,E1 21774.558,E2 21774.558} C_VEL
LIN {X 0,Y 464.99,Z 520.868,A -85,B 0,C 180,E1 21771.093,E2 21771.093} C_VEL
LIN {X 0,Y 464.959,Z 520.878,A -85,B 0,C 180,E1 21767.582,E2 21767.582} C_VEL
LIN {X 0,Y 464.967,Z 520.876,A -85,B 0,C 180,E1 21763.895,E2 21763.895} C_VEL
LIN {X 0,Y 465.007,Z 520.873,A -85,B 0,C 180,E1 21760.336,E2 21760.336} C_VEL
LIN {X 0,Y 465.007,Z 520.873,A -85,B 0,C 180,E1 21756.694,E2 21756.694} C_VEL
LIN {X 0,Y 464.974,Z 520.874,A -85,B 0,C 180,E1 21753.155,E2 21753.155} C_VEL
LIN {X 0,Y 464.98,Z 520.878,A -85,B 0,C 180,E1 21749.504,E2 21749.504} C_VEL
LIN {X 0,Y 465.009,Z 520.871,A -85,B 0,C 180,E1 21745.861,E2 21745.861} C_VEL
LIN {X 0,Y 465.049,Z 521.153,A -85,B 0,C 180,E1 21743.83,E2 21743.83} C_VEL
LIN {X 0,Y 469.937,Z 537.085,A -85,B 0,C 180,E1 21740.965,E2 21740.965} C_VEL
LIN {X 0,Y 472.9,Z 548.937,A -85,B 0,C 180,E1 21739.001,E2 21739.001} C_VEL
LIN {X 0,Y 470.946,Z 575.972,A -85,B 0,C 180,E1 21735.328,E2 21735.328} C_VEL
LIN {X 0,Y 469.197,Z 604.709,A -85,B 0,C 180,E1 21731.503,E2 21731.503} C_VEL
LIN {X 0,Y 467.868,Z 631.319,A -85,B 0,C 180,E1 21728.034,E2 21728.034} C_VEL
LIN {X 0,Y 469.133,Z 638.283,A -85,B 0,C 180,E1 21727.804,E2 21727.804} C_VEL
LIN {X 0,Y 470.875,Z 649.435,A -85,B 0,C 180,E1 21727.525,E2 21727.525} C_VEL
LIN {X 0,Y 470.071,Z 709.967,A -85,B 0,C 180,E1 21726.554,E2 21726.554} C_VEL
LIN {X 0,Y 469.053,Z 717.645,A -85,B 0,C 180,E1 21726.478,E2 21726.478} C_VEL
LIN {X 0,Y 463.001,Z 738.015,A -85,B 0,C 180,E1 21726.438,E2 21726.438} C_VEL
LIN {X 0,Y 462.217,Z 744.583,A -85,B 0,C 180,E1 21726.347,E2 21726.347} C_VEL
LIN {X 0,Y 461.933,Z 760.73,A -85,B 0,C 180,E1 21725.921,E2 21725.921} C_VEL
LIN {X 0,Y 461.434,Z 775.956,A -85,B 0,C 180,E1 21725.259,E2 21725.259} C_VEL
LIN {X 0,Y 460.792,Z 789.824,A -85,B 0,C 180,E1 21724.415,E2 21724.415} C_VEL
LIN {X 0,Y 460.025,Z 803.009,A -85,B 0,C 180,E1 21723.355,E2 21723.355} C_VEL
LIN {X 0,Y 459.25,Z 815.161,A -85,B 0,C 180,E1 21722.083,E2 21722.083} C_VEL
LIN {X 0,Y 458.585,Z 824.997,A -85,B 0,C 180,E1 21720.79,E2 21720.79} C_VEL
LIN {X 0,Y 457.895,Z 834.841,A -85,B 0,C 180,E1 21719.135,E2 21719.135} C_VEL
LIN {X 0,Y 457.37,Z 842.56,A -85,B 0,C 180,E1 21717.431,E2 21717.431} C_VEL
LIN {X 0,Y 457.014,Z 848.541,A -85,B 0,C 180,E1 21715.659,E2 21715.659} C_VEL
LIN {X 0,Y 456.771,Z 852.948,A -85,B 0,C 180,E1 21713.748,E2 21713.748} C_VEL
LIN {X 0,Y 456.636,Z 855.481,A -85,B 0,C 180,E1 21711.812,E2 21711.812} C_VEL
LIN {X 0,Y 456.59,Z 856.23,A -85,B 0,C 180,E1 21709.838,E2 21709.838} C_VEL
LIN {X 0,Y 456.625,Z 855.103,A -85,B 0,C 180,E1 21707.848,E2 21707.848} C_VEL
LIN {X 0,Y 456.736,Z 852.336,A -85,B 0,C 180,E1 21706.009,E2 21706.009} C_VEL
LIN {X 0,Y 456.951,Z 847.882,A -85,B 0,C 180,E1 21704.183,E2 21704.183} C_VEL
LIN {X 0,Y 457.291,Z 841.488,A -85,B 0,C 180,E1 21702.37,E2 21702.37} C_VEL
LIN {X 0,Y 457.78,Z 833.585,A -85,B 0,C 180,E1 21700.697,E2 21700.697} C_VEL
LIN {X 0,Y 458.394,Z 824.22,A -85,B 0,C 180,E1 21699.16,E2 21699.16} C_VEL
LIN {X 0,Y 459.107,Z 812.997,A -85,B 0,C 180,E1 21697.726,E2 21697.726} C_VEL
LIN {X 0,Y 459.796,Z 801.346,A -85,B 0,C 180,E1 21696.553,E2 21696.553} C_VEL
LIN {X 0,Y 460.547,Z 787.549,A -85,B 0,C 180,E1 21695.48,E2 21695.48} C_VEL
LIN {X 0,Y 461.143,Z 773.382,A -85,B 0,C 180,E1 21694.662,E2 21694.662} C_VEL
LIN {X 0,Y 461.588,Z 758.751,A -85,B 0,C 180,E1 21694.064,E2 21694.064} C_VEL
LIN {X 0,Y 461.855,Z 742.685,A -85,B 0,C 180,E1 21693.664,E2 21693.664} C_VEL
LIN {X 0,Y 462.793,Z 647.532,A -85,B 0,C 180,E1 21692.111,E2 21692.111} C_VEL
LIN {X 0,Y 459.925,Z 631.485,A -85,B 0,C 180,E1 21691.68,E2 21691.68} C_VEL
LIN {X 0,Y 461.334,Z 602.414,A -85,B 0,C 180,E1 21687.887,E2 21687.887} C_VEL
LIN {X 0,Y 463.102,Z 573.614,A -85,B 0,C 180,E1 21684.051,E2 21684.051} C_VEL
LIN {X 0,Y 464.691,Z 549.41,A -85,B 0,C 180,E1 21680.775,E2 21680.775} C_VEL
LIN {X 0,Y 459.978,Z 532.19,A -85,B 0,C 180,E1 21677.955,E2 21677.955} C_VEL
LIN {X 0,Y 457.023,Z 521.986,A -85,B 0,C 180,E1 21676.171,E2 21676.171} C_VEL
LIN {X 0,Y 456.999,Z 521.867,A -85,B 0,C 180,E1 21672.539,E2 21672.539} C_VEL
LIN {X 0,Y 457.032,Z 521.869,A -85,B 0,C 180,E1 21668.975,E2 21668.975} C_VEL
LIN {X 0,Y 457.03,Z 521.838,A -85,B 0,C 180,E1 21665.439,E2 21665.439} C_VEL
LIN {X 0,Y 456.993,Z 521.867,A -85,B 0,C 180,E1 21661.941,E2 21661.941} C_VEL
LIN {X 0,Y 456.993,Z 521.845,A -85,B 0,C 180,E1 21658.179,E2 21658.179} C_VEL
LIN {X 0,Y 457.042,Z 521.866,A -85,B 0,C 180,E1 21654.687,E2 21654.687} C_VEL
LIN {X 0,Y 457.023,Z 521.864,A -85,B 0,C 180,E1 21651.108,E2 21651.108} C_VEL
LIN {X 0,Y 456.995,Z 521.856,A -85,B 0,C 180,E1 21647.636,E2 21647.636} C_VEL
LIN {X 0,Y 457.021,Z 521.867,A -85,B 0,C 180,E1 21644.085,E2 21644.085} C_VEL
LIN {X 0,Y 457.065,Z 521.849,A -85,B 0,C 180,E1 21640.427,E2 21640.427} C_VEL
LIN {X 0,Y 457.018,Z 521.868,A -85,B 0,C 180,E1 21636.831,E2 21636.831} C_VEL
LIN {X 0,Y 457.003,Z 521.853,A -85,B 0,C 180,E1 21633.309,E2 21633.309} C_VEL
LIN {X 0,Y 457.034,Z 521.865,A -85,B 0,C 180,E1 21629.718,E2 21629.718} C_VEL
LIN {X 0,Y 457.057,Z 521.843,A -85,B 0,C 180,E1 21626.086,E2 21626.086} C_VEL
LIN {X 0,Y 457.017,Z 521.865,A -85,B 0,C 180,E1 21622.512,E2 21622.512} C_VEL
LIN {X 0,Y 457.012,Z 521.853,A -85,B 0,C 180,E1 21618.893,E2 21618.893} C_VEL
LIN {X 0,Y 457.042,Z 521.861,A -85,B 0,C 180,E1 21615.267,E2 21615.267} C_VEL
LIN {X 0,Y 457.056,Z 521.862,A -85,B 0,C 180,E1 21611.739,E2 21611.739} C_VEL
LIN {X 0,Y 457.017,Z 521.842,A -85,B 0,C 180,E1 21608.176,E2 21608.176} C_VEL
LIN {X 0,Y 457.02,Z 521.864,A -85,B 0,C 180,E1 21604.518,E2 21604.518} C_VEL
LIN {X 0,Y 457.063,Z 521.838,A -85,B 0,C 180,E1 21601.003,E2 21601.003} C_VEL
LIN {X 0,Y 457.055,Z 521.862,A -85,B 0,C 180,E1 21597.367,E2 21597.367} C_VEL
LIN {X 0,Y 457.022,Z 521.859,A -85,B 0,C 180,E1 21593.846,E2 21593.846} C_VEL
LIN {X 0,Y 457.031,Z 521.861,A -85,B 0,C 180,E1 21590.175,E2 21590.175} C_VEL
LIN {X 0,Y 457.071,Z 521.851,A -85,B 0,C 180,E1 21586.592,E2 21586.592} C_VEL
LIN {X 0,Y 457.062,Z 521.861,A -85,B 0,C 180,E1 21582.924,E2 21582.924} C_VEL
LIN {X 0,Y 457.029,Z 521.857,A -85,B 0,C 180,E1 21579.377,E2 21579.377} C_VEL
LIN {X 0,Y 457.036,Z 521.864,A -85,B 0,C 180,E1 21575.714,E2 21575.714} C_VEL
LIN {X 0,Y 457.076,Z 521.861,A -85,B 0,C 180,E1 21572.087,E2 21572.087} C_VEL
LIN {X 0,Y 457.066,Z 521.855,A -85,B 0,C 180,E1 21568.478,E2 21568.478} C_VEL
LIN {X 0,Y 457.037,Z 521.861,A -85,B 0,C 180,E1 21564.875,E2 21564.875} C_VEL
LIN {X 0,Y 457.037,Z 521.859,A -85,B 0,C 180,E1 21561.149,E2 21561.149} C_VEL
LIN {X 0,Y 457.071,Z 521.858,A -85,B 0,C 180,E1 21557.642,E2 21557.642} C_VEL
LIN {X 0,Y 457.076,Z 521.867,A -85,B 0,C 180,E1 21553.9,E2 21553.9} C_VEL
LIN {X 0,Y 457.053,Z 521.861,A -85,B 0,C 180,E1 21550.19,E2 21550.19} C_VEL
LIN {X 0,Y 457.075,Z 522.077,A -85,B 0,C 180,E1 21548.326,E2 21548.326} C_VEL
LIN {X 0,Y 461.583,Z 534.741,A -85,B 0,C 180,E1 21546.625,E2 21546.625} C_VEL
LIN {X 0,Y 468.998,Z 556.285,A -85,B 0,C 180,E1 21543.972,E2 21543.972} C_VEL
LIN {X 0,Y 466.04,Z 598.944,A -85,B 0,C 180,E1 21540.204,E2 21540.204} C_VEL
LIN {X 0,Y 465.037,Z 616.444,A -85,B 0,C 180,E1 21538.716,E2 21538.716} C_VEL
LIN {X 0,Y 467.311,Z 636.085,A -85,B 0,C 180,E1 21538.273,E2 21538.273} C_VEL
LIN {X 0,Y 465.154,Z 819.326,A -85,B 0,C 180,E1 21535.405,E2 21535.405} C_VEL
LIN {X 0,Y 464.46,Z 838.164,A -85,B 0,C 180,E1 21534.89,E2 21534.89} C_VEL
LIN {X 0,Y 463.555,Z 856.371,A -85,B 0,C 180,E1 21534.163,E2 21534.163} C_VEL
LIN {X 0,Y 462.552,Z 873.808,A -85,B 0,C 180,E1 21533.234,E2 21533.234} C_VEL
LIN {X 0,Y 461.41,Z 890.824,A -85,B 0,C 180,E1 21532.084,E2 21532.084} C_VEL
LIN {X 0,Y 460.26,Z 907.637,A -85,B 0,C 180,E1 21530.671,E2 21530.671} C_VEL
LIN {X 0,Y 459.18,Z 923.079,A -85,B 0,C 180,E1 21529.086,E2 21529.086} C_VEL
LIN {X 0,Y 458.24,Z 936.743,A -85,B 0,C 180,E1 21527.393,E2 21527.393} C_VEL
LIN {X 0,Y 457.446,Z 949.665,A -85,B 0,C 180,E1 21525.466,E2 21525.466} C_VEL
LIN {X 0,Y 456.855,Z 960.997,A -85,B 0,C 180,E1 21523.415,E2 21523.415} C_VEL
LIN {X 0,Y 456.471,Z 970.717,A -85,B 0,C 180,E1 21521.242,E2 21521.242} C_VEL
LIN {X 0,Y 456.266,Z 978.406,A -85,B 0,C 180,E1 21519.079,E2 21519.079} C_VEL
LIN {X 0,Y 456.189,Z 984.572,A -85,B 0,C 180,E1 21516.798,E2 21516.798} C_VEL
LIN {X 0,Y 456.201,Z 988.884,A -85,B 0,C 180,E1 21514.527,E2 21514.527} C_VEL
LIN {X 0,Y 456.234,Z 991.435,A -85,B 0,C 180,E1 21512.262,E2 21512.262} C_VEL
LIN {X 0,Y 456.255,Z 992.274,A -85,B 0,C 180,E1 21510.002,E2 21510.002} C_VEL
LIN {X 0,Y 456.238,Z 991.405,A -85,B 0,C 180,E1 21507.741,E2 21507.741} C_VEL
LIN {X 0,Y 456.209,Z 988.825,A -85,B 0,C 180,E1 21505.477,E2 21505.477} C_VEL
LIN {X 0,Y 456.199,Z 984.484,A -85,B 0,C 180,E1 21503.205,E2 21503.205} C_VEL
LIN {X 0,Y 456.276,Z 978.279,A -85,B 0,C 180,E1 21500.924,E2 21500.924} C_VEL
LIN {X 0,Y 456.481,Z 970.542,A -85,B 0,C 180,E1 21498.761,E2 21498.761} C_VEL
LIN {X 0,Y 456.86,Z 960.766,A -85,B 0,C 180,E1 21496.589,E2 21496.589} C_VEL
LIN {X 0,Y 457.443,Z 949.369,A -85,B 0,C 180,E1 21494.537,E2 21494.537} C_VEL
LIN {X 0,Y 458.225,Z 936.373,A -85,B 0,C 180,E1 21492.609,E2 21492.609} C_VEL
LIN {X 0,Y 459.152,Z 922.733,A -85,B 0,C 180,E1 21490.924,E2 21490.924} C_VEL
LIN {X 0,Y 460.181,Z 907.884,A -85,B 0,C 180,E1 21489.395,E2 21489.395} C_VEL
LIN {X 0,Y 461.247,Z 892.117,A -85,B 0,C 180,E1 21488.052,E2 21488.052} C_VEL
LIN {X 0,Y 462.448,Z 874.346,A -85,B 0,C 180,E1 21486.831,E2 21486.831} C_VEL
LIN {X 0,Y 463.477,Z 856.59,A -85,B 0,C 180,E1 21485.874,E2 21485.874} C_VEL
LIN {X 0,Y 464.391,Z 838.329,A -85,B 0,C 180,E1 21485.137,E2 21485.137} C_VEL
LIN {X 0,Y 465.096,Z 819.523,A -85,B 0,C 180,E1 21484.616,E2 21484.616} C_VEL
LIN {X 0,Y 465.705,Z 770.6,A -85,B 0,C 180,E1 21483.836,E2 21483.836} C_VEL
LIN {X 0,Y 467.138,Z 633.066,A -85,B 0,C 180,E1 21481.671,E2 21481.671} C_VEL
LIN {X 0,Y 465.068,Z 615.859,A -85,B 0,C 180,E1 21481.233,E2 21481.233} C_VEL
LIN {X 0,Y 468.123,Z 572.271,A -85,B 0,C 180,E1 21477.368,E2 21477.368} C_VEL
LIN {X 0,Y 469.3,Z 556.546,A -85,B 0,C 180,E1 21475.927,E2 21475.927} C_VEL
LIN {X 0,Y 462.933,Z 537.559,A -85,B 0,C 180,E1 21473.462,E2 21473.462} C_VEL
LIN {X 0,Y 457.073,Z 522.076,A -85,B 0,C 180,E1 21471.165,E2 21471.165} C_VEL
LIN {X 0,Y 457.035,Z 521.866,A -85,B 0,C 180,E1 21467.498,E2 21467.498} C_VEL
LIN {X 0,Y 457.058,Z 521.862,A -85,B 0,C 180,E1 21463.905,E2 21463.905} C_VEL
LIN {X 0,Y 457.081,Z 521.865,A -85,B 0,C 180,E1 21460.189,E2 21460.189} C_VEL
LIN {X 0,Y 457.043,Z 521.866,A -85,B 0,C 180,E1 21456.516,E2 21456.516} C_VEL
LIN {X 0,Y 457.018,Z 521.865,A -85,B 0,C 180,E1 21452.859,E2 21452.859} C_VEL
LIN {X 0,Y 457.023,Z 521.864,A -85,B 0,C 180,E1 21449.201,E2 21449.201} C_VEL
LIN {X 0,Y 457.061,Z 521.866,A -85,B 0,C 180,E1 21445.667,E2 21445.667} C_VEL
LIN {X 0,Y 457.028,Z 521.864,A -85,B 0,C 180,E1 21442.104,E2 21442.104} C_VEL
LIN {X 0,Y 457.001,Z 521.861,A -85,B 0,C 180,E1 21438.496,E2 21438.496} C_VEL
LIN {X 0,Y 457.003,Z 521.854,A -85,B 0,C 180,E1 21434.831,E2 21434.831} C_VEL
LIN {X 0,Y 457.05,Z 521.864,A -85,B 0,C 180,E1 21431.355,E2 21431.355} C_VEL
LIN {X 0,Y 457.022,Z 521.866,A -85,B 0,C 180,E1 21427.669,E2 21427.669} C_VEL
LIN {X 0,Y 456.997,Z 521.857,A -85,B 0,C 180,E1 21424.14,E2 21424.14} C_VEL
LIN {X 0,Y 457.015,Z 521.857,A -85,B 0,C 180,E1 21420.501,E2 21420.501} C_VEL
LIN {X 0,Y 457.061,Z 521.864,A -85,B 0,C 180,E1 21416.99,E2 21416.99} C_VEL
LIN {X 0,Y 457.034,Z 521.864,A -85,B 0,C 180,E1 21413.341,E2 21413.341} C_VEL
LIN {X 0,Y 457.015,Z 521.86,A -85,B 0,C 180,E1 21409.792,E2 21409.792} C_VEL
LIN {X 0,Y 457.038,Z 521.856,A -85,B 0,C 180,E1 21406.204,E2 21406.204} C_VEL
LIN {X 0,Y 457.072,Z 521.854,A -85,B 0,C 180,E1 21402.692,E2 21402.692} C_VEL
LIN {X 0,Y 457.041,Z 521.859,A -85,B 0,C 180,E1 21399.072,E2 21399.072} C_VEL
LIN {X 0,Y 457.031,Z 521.859,A -85,B 0,C 180,E1 21395.438,E2 21395.438} C_VEL
LIN {X 0,Y 457.053,Z 521.866,A -85,B 0,C 180,E1 21391.801,E2 21391.801} C_VEL
LIN {X 0,Y 457.079,Z 521.858,A -85,B 0,C 180,E1 21388.184,E2 21388.184} C_VEL
LIN {X 0,Y 457.088,Z 522.034,A -85,B 0,C 180,E1 21384.511,E2 21384.511} C_VEL
LIN {X 0,Y 461.724,Z 536.911,A -85,B 0,C 180,E1 21381.732,E2 21381.732} C_VEL
LIN {X 0,Y 465.567,Z 551.089,A -85,B 0,C 180,E1 21379.29,E2 21379.29} C_VEL
LIN {X 0,Y 463.477,Z 578.164,A -85,B 0,C 180,E1 21375.559,E2 21375.559} C_VEL
LIN {X 0,Y 461.597,Z 606.916,A -85,B 0,C 180,E1 21371.675,E2 21371.675} C_VEL
LIN {X 0,Y 460.288,Z 631.326,A -85,B 0,C 180,E1 21368.451,E2 21368.451} C_VEL
LIN {X 0,Y 463.558,Z 650.154,A -85,B 0,C 180,E1 21367.915,E2 21367.915} C_VEL
LIN {X 0,Y 462.217,Z 744.583,A -85,B 0,C 180,E1 21366.347,E2 21366.347} C_VEL
LIN {X 0,Y 460.878,Z 753.3,A -85,B 0,C 180,E1 21366.211,E2 21366.211} C_VEL
LIN {X 0,Y 455.716,Z 769.069,A -85,B 0,C 180,E1 21365.912,E2 21365.912} C_VEL
LIN {X 0,Y 454.101,Z 776.312,A -85,B 0,C 180,E1 21365.635,E2 21365.635} C_VEL
LIN {X 0,Y 453.927,Z 778.351,A -85,B 0,C 180,E1 21365.529,E2 21365.529} C_VEL
LIN {X 0,Y 453.202,Z 792.466,A -85,B 0,C 180,E1 21364.621,E2 21364.621} C_VEL
LIN {X 0,Y 452.378,Z 805.303,A -85,B 0,C 180,E1 21363.537,E2 21363.537} C_VEL
LIN {X 0,Y 451.528,Z 817.722,A -85,B 0,C 180,E1 21362.181,E2 21362.181} C_VEL
LIN {X 0,Y 450.714,Z 828.42,A -85,B 0,C 180,E1 21360.674,E2 21360.674} C_VEL
LIN {X 0,Y 450.046,Z 837.139,A -85,B 0,C 180,E1 21359.109,E2 21359.109} C_VEL
LIN {X 0,Y 449.475,Z 844.986,A -85,B 0,C 180,E1 21357.27,E2 21357.27} C_VEL
LIN {X 0,Y 449.075,Z 850.997,A -85,B 0,C 180,E1 21355.304,E2 21355.304} C_VEL
LIN {X 0,Y 448.837,Z 854.854,A -85,B 0,C 180,E1 21353.393,E2 21353.393} C_VEL
LIN {X 0,Y 448.715,Z 857.001,A -85,B 0,C 180,E1 21351.431,E2 21351.431} C_VEL
LIN {X 0,Y 448.677,Z 857.311,A -85,B 0,C 180,E1 21349.389,E2 21349.389} C_VEL
LIN {X 0,Y 448.728,Z 855.928,A -85,B 0,C 180,E1 21347.503,E2 21347.503} C_VEL
LIN {X 0,Y 448.887,Z 852.635,A -85,B 0,C 180,E1 21345.5,E2 21345.5} C_VEL
LIN {X 0,Y 449.148,Z 847.714,A -85,B 0,C 180,E1 21343.646,E2 21343.646} C_VEL
LIN {X 0,Y 449.55,Z 841.162,A -85,B 0,C 180,E1 21341.868,E2 21341.868} C_VEL
LIN {X 0,Y 450.148,Z 832.477,A -85,B 0,C 180,E1 21340.104,E2 21340.104} C_VEL
LIN {X 0,Y 450.842,Z 822.464,A -85,B 0,C 180,E1 21338.543,E2 21338.543} C_VEL
LIN {X 0,Y 451.59,Z 811.405,A -85,B 0,C 180,E1 21337.184,E2 21337.184} C_VEL
LIN {X 0,Y 452.386,Z 798.674,A -85,B 0,C 180,E1 21335.961,E2 21335.961} C_VEL
LIN {X 0,Y 453.088,Z 785.624,A -85,B 0,C 180,E1 21334.999,E2 21334.999} C_VEL
LIN {X 0,Y 453.705,Z 771.195,A -85,B 0,C 180,E1 21334.2,E2 21334.2} C_VEL
LIN {X 0,Y 454.167,Z 755.215,A -85,B 0,C 180,E1 21333.599,E2 21333.599} C_VEL
LIN {X 0,Y 454.423,Z 736.562,A -85,B 0,C 180,E1 21333.211,E2 21333.211} C_VEL
LIN {X 0,Y 455.369,Z 648.668,A -85,B 0,C 180,E1 21331.755,E2 21331.755} C_VEL
LIN {X 0,Y 452.28,Z 631.154,A -85,B 0,C 180,E1 21331.265,E2 21331.265} C_VEL
LIN {X 0,Y 453.847,Z 601.614,A -85,B 0,C 180,E1 21327.347,E2 21327.347} C_VEL
LIN {X 0,Y 455.735,Z 572.791,A -85,B 0,C 180,E1 21323.448,E2 21323.448} C_VEL
LIN {X 0,Y 457.147,Z 551.652,A -85,B 0,C 180,E1 21320.548,E2 21320.548} C_VEL
LIN {X 0,Y 452.327,Z 534.04,A -85,B 0,C 180,E1 21317.618,E2 21317.618} C_VEL
LIN {X 0,Y 449.123,Z 522.969,A -85,B 0,C 180,E1 21315.657,E2 21315.657} C_VEL
LIN {X 0,Y 449.065,Z 522.858,A -85,B 0,C 180,E1 21312.106,E2 21312.106} C_VEL
LIN {X 0,Y 449.059,Z 522.858,A -85,B 0,C 180,E1 21308.446,E2 21308.446} C_VEL
LIN {X 0,Y 449.099,Z 522.833,A -85,B 0,C 180,E1 21304.976,E2 21304.976} C_VEL
LIN {X 0,Y 449.091,Z 522.836,A -85,B 0,C 180,E1 21301.308,E2 21301.308} C_VEL
LIN {X 0,Y 449.053,Z 522.84,A -85,B 0,C 180,E1 21297.699,E2 21297.699} C_VEL
LIN {X 0,Y 449.056,Z 522.854,A -85,B 0,C 180,E1 21293.926,E2 21293.926} C_VEL
LIN {X 0,Y 449.081,Z 522.858,A -85,B 0,C 180,E1 21290.285,E2 21290.285} C_VEL
LIN {X 0,Y 449.109,Z 522.841,A -85,B 0,C 180,E1 21286.711,E2 21286.711} C_VEL
LIN {X 0,Y 449.071,Z 522.856,A -85,B 0,C 180,E1 21283.092,E2 21283.092} C_VEL
LIN {X 0,Y 449.061,Z 522.852,A -85,B 0,C 180,E1 21279.414,E2 21279.414} C_VEL
LIN {X 0,Y 449.09,Z 522.846,A -85,B 0,C 180,E1 21275.842,E2 21275.842} C_VEL
LIN {X 0,Y 449.121,Z 522.844,A -85,B 0,C 180,E1 21272.146,E2 21272.146} C_VEL
LIN {X 0,Y 449.08,Z 522.855,A -85,B 0,C 180,E1 21268.6,E2 21268.6} C_VEL
LIN {X 0,Y 449.069,Z 522.841,A -85,B 0,C 180,E1 21265.023,E2 21265.023} C_VEL
LIN {X 0,Y 449.098,Z 522.853,A -85,B 0,C 180,E1 21261.416,E2 21261.416} C_VEL
LIN {X 0,Y 449.124,Z 522.828,A -85,B 0,C 180,E1 21257.758,E2 21257.758} C_VEL
LIN {X 0,Y 449.086,Z 522.852,A -85,B 0,C 180,E1 21254.177,E2 21254.177} C_VEL
LIN {X 0,Y 449.075,Z 522.845,A -85,B 0,C 180,E1 21250.52,E2 21250.52} C_VEL
LIN {X 0,Y 449.091,Z 522.846,A -85,B 0,C 180,E1 21246.823,E2 21246.823} C_VEL
LIN {X 0,Y 449.128,Z 522.846,A -85,B 0,C 180,E1 21243.191,E2 21243.191} C_VEL
LIN {X 0,Y 449.11,Z 522.83,A -85,B 0,C 180,E1 21239.49,E2 21239.49} C_VEL
LIN {X 0,Y 449.084,Z 522.855,A -85,B 0,C 180,E1 21235.855,E2 21235.855} C_VEL
LIN {X 0,Y 449.084,Z 522.834,A -85,B 0,C 180,E1 21232.066,E2 21232.066} C_VEL
LIN {X 0,Y 449.114,Z 522.852,A -85,B 0,C 180,E1 21228.442,E2 21228.442} C_VEL
LIN {X 0,Y 449.14,Z 522.835,A -85,B 0,C 180,E1 21224.771,E2 21224.771} C_VEL
LIN {X 0,Y 449.112,Z 522.856,A -85,B 0,C 180,E1 21221.032,E2 21221.032} C_VEL
LIN {X 0,Y 449.09,Z 522.849,A -85,B 0,C 180,E1 21217.346,E2 21217.346} C_VEL
LIN {X 0,Y 449.095,Z 522.84,A -85,B 0,C 180,E1 21213.559,E2 21213.559} C_VEL
LIN {X 0,Y 449.129,Z 522.846,A -85,B 0,C 180,E1 21209.941,E2 21209.941} C_VEL
LIN {X 0,Y 449.137,Z 522.851,A -85,B 0,C 180,E1 21206.183,E2 21206.183} C_VEL
LIN {X 0,Y 449.123,Z 522.856,A -85,B 0,C 180,E1 21202.411,E2 21202.411} C_VEL
LIN {X 0,Y 449.101,Z 522.856,A -85,B 0,C 180,E1 21198.776,E2 21198.776} C_VEL
LIN {X 0,Y 449.105,Z 522.847,A -85,B 0,C 180,E1 21195.068,E2 21195.068} C_VEL
LIN {X 0,Y 449.139,Z 522.853,A -85,B 0,C 180,E1 21191.387,E2 21191.387} C_VEL
LIN {X 0,Y 449.147,Z 523.118,A -85,B 0,C 180,E1 21188.884,E2 21188.884} C_VEL
LIN {X 0,Y 457.168,Z 545.618,A -85,B 0,C 180,E1 21185.881,E2 21185.881} C_VEL
LIN {X 0,Y 461.656,Z 559.135,A -85,B 0,C 180,E1 21184.216,E2 21184.216} C_VEL
LIN {X 0,Y 458.319,Z 603.981,A -85,B 0,C 180,E1 21180.188,E2 21180.188} C_VEL
LIN {X 0,Y 457.55,Z 616.152,A -85,B 0,C 180,E1 21179.131,E2 21179.131} C_VEL
LIN {X 0,Y 459.914,Z 636.992,A -85,B 0,C 180,E1 21178.641,E2 21178.641} C_VEL
LIN {X 0,Y 457.656,Z 818.598,A -85,B 0,C 180,E1 21175.761,E2 21175.761} C_VEL
LIN {X 0,Y 456.923,Z 837.446,A -85,B 0,C 180,E1 21175.239,E2 21175.239} C_VEL
LIN {X 0,Y 455.979,Z 855.318,A -85,B 0,C 180,E1 21174.518,E2 21174.518} C_VEL
LIN {X 0,Y 454.921,Z 872.745,A -85,B 0,C 180,E1 21173.578,E2 21173.578} C_VEL
LIN {X 0,Y 453.719,Z 889.797,A -85,B 0,C 180,E1 21172.41,E2 21172.41} C_VEL
LIN {X 0,Y 452.49,Z 906.625,A -85,B 0,C 180,E1 21170.975,E2 21170.975} C_VEL
LIN {X 0,Y 451.375,Z 921.69,A -85,B 0,C 180,E1 21169.407,E2 21169.407} C_VEL
LIN {X 0,Y 450.384,Z 935.265,A -85,B 0,C 180,E1 21167.707,E2 21167.707} C_VEL
LIN {X 0,Y 449.587,Z 947.473,A -85,B 0,C 180,E1 21165.876,E2 21165.876} C_VEL
LIN {X 0,Y 448.951,Z 958.802,A -85,B 0,C 180,E1 21163.829,E2 21163.829} C_VEL
LIN {X 0,Y 448.54,Z 968.388,A -85,B 0,C 180,E1 21161.704,E2 21161.704} C_VEL
LIN {X 0,Y 448.329,Z 976.342,A -85,B 0,C 180,E1 21159.5,E2 21159.5} C_VEL
LIN {X 0,Y 448.244,Z 982.446,A -85,B 0,C 180,E1 21157.306,E2 21157.306} C_VEL
LIN {X 0,Y 448.259,Z 986.86,A -85,B 0,C 180,E1 21155.12,E2 21155.12} C_VEL
LIN {X 0,Y 448.305,Z 989.798,A -85,B 0,C 180,E1 21152.814,E2 21152.814} C_VEL
LIN {X 0,Y 448.335,Z 991.009,A -85,B 0,C 180,E1 21150.513,E2 21150.513} C_VEL
LIN {X 0,Y 448.331,Z 990.518,A -85,B 0,C 180,E1 21148.213,E2 21148.213} C_VEL
LIN {X 0,Y 448.295,Z 988.314,A -85,B 0,C 180,E1 21145.909,E2 21145.909} C_VEL
LIN {X 0,Y 448.261,Z 984.352,A -85,B 0,C 180,E1 21143.599,E2 21143.599} C_VEL
LIN {X 0,Y 448.294,Z 978.532,A -85,B 0,C 180,E1 21141.279,E2 21141.279} C_VEL
LIN {X 0,Y 448.464,Z 971.2,A -85,B 0,C 180,E1 21139.078,E2 21139.078} C_VEL
LIN {X 0,Y 448.8,Z 961.878,A -85,B 0,C 180,E1 21136.868,E2 21136.868} C_VEL
LIN {X 0,Y 449.357,Z 951.027,A -85,B 0,C 180,E1 21134.781,E2 21134.781} C_VEL
LIN {X 0,Y 450.117,Z 938.654,A -85,B 0,C 180,E1 21132.819,E2 21132.819} C_VEL
LIN {X 0,Y 451.101,Z 924.713,A -85,B 0,C 180,E1 21130.988,E2 21130.988} C_VEL
LIN {X 0,Y 452.187,Z 910.006,A -85,B 0,C 180,E1 21129.385,E2 21129.385} C_VEL
LIN {X 0,Y 453.374,Z 893.616,A -85,B 0,C 180,E1 21127.917,E2 21127.917} C_VEL
LIN {X 0,Y 454.619,Z 876.518,A -85,B 0,C 180,E1 21126.683,E2 21126.683} C_VEL
LIN {X 0,Y 455.707,Z 859.227,A -85,B 0,C 180,E1 21125.692,E2 21125.692} C_VEL
LIN {X 0,Y 456.703,Z 840.927,A -85,B 0,C 180,E1 21124.897,E2 21124.897} C_VEL
LIN {X 0,Y 457.519,Z 822.068,A -85,B 0,C 180,E1 21124.326,E2 21124.326} C_VEL
LIN {X 0,Y 457.992,Z 796.274,A -85,B 0,C 180,E1 21123.863,E2 21123.863} C_VEL
LIN {X 0,Y 459.837,Z 634.131,A -85,B 0,C 180,E1 21121.28,E2 21121.28} C_VEL
LIN {X 0,Y 457.682,Z 616.069,A -85,B 0,C 180,E1 21120.814,E2 21120.814} C_VEL
LIN {X 0,Y 460.944,Z 573.334,A -85,B 0,C 180,E1 21116.943,E2 21116.943} C_VEL
LIN {X 0,Y 462.04,Z 559.215,A -85,B 0,C 180,E1 21115.616,E2 21115.616} C_VEL
LIN {X 0,Y 455.912,Z 540.924,A -85,B 0,C 180,E1 21113.176,E2 21113.176} C_VEL
LIN {X 0,Y 450.333,Z 526.262,A -85,B 0,C 180,E1 21110.995,E2 21110.995} C_VEL
LIN {X 0,Y 449.165,Z 523.015,A -85,B 0,C 180,E1 21110.423,E2 21110.423} C_VEL
LIN {X 0,Y 449.117,Z 522.849,A -85,B 0,C 180,E1 21106.717,E2 21106.717} C_VEL
LIN {X 0,Y 449.091,Z 522.858,A -85,B 0,C 180,E1 21103.099,E2 21103.099} C_VEL
LIN {X 0,Y 449.09,Z 522.849,A -85,B 0,C 180,E1 21099.385,E2 21099.385} C_VEL
LIN {X 0,Y 449.122,Z 522.845,A -85,B 0,C 180,E1 21095.838,E2 21095.838} C_VEL
LIN {X 0,Y 449.121,Z 522.844,A -85,B 0,C 180,E1 21092.146,E2 21092.146} C_VEL
LIN {X 0,Y 449.079,Z 522.851,A -85,B 0,C 180,E1 21088.6,E2 21088.6} C_VEL
LIN {X 0,Y 449.072,Z 522.853,A -85,B 0,C 180,E1 21084.885,E2 21084.885} C_VEL
LIN {X 0,Y 449.095,Z 522.856,A -85,B 0,C 180,E1 21081.278,E2 21081.278} C_VEL
LIN {X 0,Y 449.114,Z 522.85,A -85,B 0,C 180,E1 21077.624,E2 21077.624} C_VEL
LIN {X 0,Y 449.067,Z 522.842,A -85,B 0,C 180,E1 21074.045,E2 21074.045} C_VEL
LIN {X 0,Y 449.054,Z 522.851,A -85,B 0,C 180,E1 21070.39,E2 21070.39} C_VEL
LIN {X 0,Y 449.077,Z 522.857,A -85,B 0,C 180,E1 21066.777,E2 21066.777} C_VEL
LIN {X 0,Y 449.113,Z 522.848,A -85,B 0,C 180,E1 21063.19,E2 21063.19} C_VEL
LIN {X 0,Y 449.078,Z 522.843,A -85,B 0,C 180,E1 21059.617,E2 21059.617} C_VEL
LIN {X 0,Y 449.069,Z 522.852,A -85,B 0,C 180,E1 21056.042,E2 21056.042} C_VEL
LIN {X 0,Y 449.1,Z 522.854,A -85,B 0,C 180,E1 21052.452,E2 21052.452} C_VEL
LIN {X 0,Y 449.129,Z 522.853,A -85,B 0,C 180,E1 21048.832,E2 21048.832} C_VEL
LIN {X 0,Y 449.099,Z 522.85,A -85,B 0,C 180,E1 21045.165,E2 21045.165} C_VEL
LIN {X 0,Y 449.087,Z 522.852,A -85,B 0,C 180,E1 21041.504,E2 21041.504} C_VEL
LIN {X 0,Y 449.096,Z 522.856,A -85,B 0,C 180,E1 21037.76,E2 21037.76} C_VEL
LIN {X 0,Y 449.129,Z 522.852,A -85,B 0,C 180,E1 21034.129,E2 21034.129} C_VEL
LIN {X 0,Y 449.139,Z 522.846,A -85,B 0,C 180,E1 21030.382,E2 21030.382} C_VEL
LIN {X 0,Y 449.121,Z 522.854,A -85,B 0,C 180,E1 21026.64,E2 21026.64} C_VEL
LIN {X 0,Y 449.143,Z 523.144,A -85,B 0,C 180,E1 21025.16,E2 21025.16} C_VEL
LIN {X 0,Y 454.057,Z 538.418,A -85,B 0,C 180,E1 21022.227,E2 21022.227} C_VEL
LIN {X 0,Y 458.199,Z 553.774,A -85,B 0,C 180,E1 21019.519,E2 21019.519} C_VEL
LIN {X 0,Y 456.015,Z 580.399,A -85,B 0,C 180,E1 21015.793,E2 21015.793} C_VEL
LIN {X 0,Y 454.028,Z 608.83,A -85,B 0,C 180,E1 21011.897,E2 21011.897} C_VEL
LIN {X 0,Y 452.729,Z 630.797,A -85,B 0,C 180,E1 21008.938,E2 21008.938} C_VEL
LIN {X 0,Y 453.503,Z 635.295,A -85,B 0,C 180,E1 21008.757,E2 21008.757} C_VEL
LIN {X 0,Y 456.264,Z 651.514,A -85,B 0,C 180,E1 21008.31,E2 21008.31} C_VEL
LIN {X 0,Y 454.754,Z 750.822,A -85,B 0,C 180,E1 21006.605,E2 21006.605} C_VEL
LIN {X 0,Y 454.378,Z 766.522,A -85,B 0,C 180,E1 21006.094,E2 21006.094} C_VEL
LIN {X 0,Y 453.927,Z 778.351,A -85,B 0,C 180,E1 21005.529,E2 21005.529} C_VEL
LIN {X 0,Y 452.659,Z 785.493,A -85,B 0,C 180,E1 21005.155,E2 21005.155} C_VEL
LIN {X 0,Y 447.385,Z 799.045,A -85,B 0,C 180,E1 21004.401,E2 21004.401} C_VEL
LIN {X 0,Y 445.017,Z 806.353,A -85,B 0,C 180,E1 21003.84,E2 21003.84} C_VEL
LIN {X 0,Y 444.641,Z 808.936,A -85,B 0,C 180,E1 21003.591,E2 21003.591} C_VEL
LIN {X 0,Y 443.782,Z 820.297,A -85,B 0,C 180,E1 21002.269,E2 21002.269} C_VEL
LIN {X 0,Y 442.941,Z 830.669,A -85,B 0,C 180,E1 21000.744,E2 21000.744} C_VEL
LIN {X 0,Y 442.199,Z 839.44,A -85,B 0,C 180,E1 20999.082,E2 20999.082} C_VEL
LIN {X 0,Y 441.64,Z 846.47,A -85,B 0,C 180,E1 20997.356,E2 20997.356} C_VEL
LIN {X 0,Y 441.206,Z 852.39,A -85,B 0,C 180,E1 20995.356,E2 20995.356} C_VEL
LIN {X 0,Y 440.939,Z 856.201,A -85,B 0,C 180,E1 20993.376,E2 20993.376} C_VEL
LIN {X 0,Y 440.805,Z 858.218,A -85,B 0,C 180,E1 20991.416,E2 20991.416} C_VEL
LIN {X 0,Y 440.766,Z 858.476,A -85,B 0,C 180,E1 20989.32,E2 20989.32} C_VEL
LIN {X 0,Y 440.821,Z 857.042,A -85,B 0,C 180,E1 20987.418,E2 20987.418} C_VEL
LIN {X 0,Y 440.999,Z 853.711,A -85,B 0,C 180,E1 20985.38,E2 20985.38} C_VEL
LIN {X 0,Y 441.315,Z 848.341,A -85,B 0,C 180,E1 20983.359,E2 20983.359} C_VEL
LIN {X 0,Y 441.745,Z 841.879,A -85,B 0,C 180,E1 20981.619,E2 20981.619} C_VEL
LIN {X 0,Y 442.372,Z 833.443,A -85,B 0,C 180,E1 20979.889,E2 20979.889} C_VEL
LIN {X 0,Y 443.115,Z 823.396,A -85,B 0,C 180,E1 20978.301,E2 20978.301} C_VEL
LIN {X 0,Y 443.911,Z 812.306,A -85,B 0,C 180,E1 20976.919,E2 20976.919} C_VEL
LIN {X 0,Y 444.756,Z 799.563,A -85,B 0,C 180,E1 20975.675,E2 20975.675} C_VEL
LIN {X 0,Y 445.55,Z 785.53,A -85,B 0,C 180,E1 20974.632,E2 20974.632} C_VEL
LIN {X 0,Y 446.175,Z 771.433,A -85,B 0,C 180,E1 20973.853,E2 20973.853} C_VEL
LIN {X 0,Y 446.656,Z 755.564,A -85,B 0,C 180,E1 20973.252,E2 20973.252} C_VEL
LIN {X 0,Y 446.935,Z 735.956,A -85,B 0,C 180,E1 20972.843,E2 20972.843} C_VEL
LIN {X 0,Y 447.938,Z 649.723,A -85,B 0,C 180,E1 20971.389,E2 20971.389} C_VEL
LIN {X 0,Y 444.65,Z 631.115,A -85,B 0,C 180,E1 20970.868,E2 20970.868} C_VEL
LIN {X 0,Y 446.323,Z 601.741,A -85,B 0,C 180,E1 20966.917,E2 20966.917} C_VEL
LIN {X 0,Y 448.258,Z 573.751,A -85,B 0,C 180,E1 20963.081,E2 20963.081} C_VEL
LIN {X 0,Y 449.719,Z 554.442,A -85,B 0,C 180,E1 20960.401,E2 20960.401} C_VEL
LIN {X 0,Y 445.124,Z 537.498,A -85,B 0,C 180,E1 20957.546,E2 20957.546} C_VEL
LIN {X 0,Y 441.17,Z 523.975,A -85,B 0,C 180,E1 20955.127,E2 20955.127} C_VEL
LIN {X 0,Y 441.17,Z 523.847,A -85,B 0,C 180,E1 20951.501,E2 20951.501} C_VEL
LIN {X 0,Y 441.125,Z 523.832,A -85,B 0,C 180,E1 20947.898,E2 20947.898} C_VEL
LIN {X 0,Y 441.117,Z 523.845,A -85,B 0,C 180,E1 20944.141,E2 20944.141} C_VEL
LIN {X 0,Y 441.127,Z 523.812,A -85,B 0,C 180,E1 20940.503,E2 20940.503} C_VEL
LIN {X 0,Y 441.171,Z 523.83,A -85,B 0,C 180,E1 20936.895,E2 20936.895} C_VEL
LIN {X 0,Y 441.145,Z 523.836,A -85,B 0,C 180,E1 20933.138,E2 20933.138} C_VEL
LIN {X 0,Y 441.119,Z 523.847,A -85,B 0,C 180,E1 20929.592,E2 20929.592} C_VEL
LIN {X 0,Y 441.129,Z 523.843,A -85,B 0,C 180,E1 20925.908,E2 20925.908} C_VEL
LIN {X 0,Y 441.17,Z 523.829,A -85,B 0,C 180,E1 20922.308,E2 20922.308} C_VEL
LIN {X 0,Y 441.152,Z 523.841,A -85,B 0,C 180,E1 20918.723,E2 20918.723} C_VEL
LIN {X 0,Y 441.126,Z 523.836,A -85,B 0,C 180,E1 20915.095,E2 20915.095} C_VEL
LIN {X 0,Y 441.13,Z 523.843,A -85,B 0,C 180,E1 20911.269,E2 20911.269} C_VEL
LIN {X 0,Y 441.161,Z 523.828,A -85,B 0,C 180,E1 20907.686,E2 20907.686} C_VEL
LIN {X 0,Y 441.187,Z 523.832,A -85,B 0,C 180,E1 20903.933,E2 20903.933} C_VEL
LIN {X 0,Y 441.151,Z 523.844,A -85,B 0,C 180,E1 20900.29,E2 20900.29} C_VEL
LIN {X 0,Y 441.132,Z 523.824,A -85,B 0,C 180,E1 20896.594,E2 20896.594} C_VEL
LIN {X 0,Y 441.142,Z 523.843,A -85,B 0,C 180,E1 20892.834,E2 20892.834} C_VEL
LIN {X 0,Y 441.179,Z 523.813,A -85,B 0,C 180,E1 20889.26,E2 20889.26} C_VEL
LIN {X 0,Y 441.175,Z 523.838,A -85,B 0,C 180,E1 20885.593,E2 20885.593} C_VEL
LIN {X 0,Y 441.146,Z 523.835,A -85,B 0,C 180,E1 20881.949,E2 20881.949} C_VEL
LIN {X 0,Y 441.142,Z 523.837,A -85,B 0,C 180,E1 20878.147,E2 20878.147} C_VEL
LIN {X 0,Y 441.157,Z 523.835,A -85,B 0,C 180,E1 20874.407,E2 20874.407} C_VEL
LIN {X 0,Y 441.191,Z 523.831,A -85,B 0,C 180,E1 20870.741,E2 20870.741} C_VEL
LIN {X 0,Y 441.182,Z 523.836,A -85,B 0,C 180,E1 20867.023,E2 20867.023} C_VEL
LIN {X 0,Y 441.154,Z 523.837,A -85,B 0,C 180,E1 20863.407,E2 20863.407} C_VEL
LIN {X 0,Y 441.152,Z 523.834,A -85,B 0,C 180,E1 20859.71,E2 20859.71} C_VEL
LIN {X 0,Y 441.18,Z 523.841,A -85,B 0,C 180,E1 20856.067,E2 20856.067} C_VEL
LIN {X 0,Y 441.203,Z 523.833,A -85,B 0,C 180,E1 20852.318,E2 20852.318} C_VEL
LIN {X 0,Y 441.181,Z 523.832,A -85,B 0,C 180,E1 20848.584,E2 20848.584} C_VEL
LIN {X 0,Y 441.16,Z 523.837,A -85,B 0,C 180,E1 20844.853,E2 20844.853} C_VEL
LIN {X 0,Y 441.158,Z 523.836,A -85,B 0,C 180,E1 20841.112,E2 20841.112} C_VEL
LIN {X 0,Y 441.182,Z 523.837,A -85,B 0,C 180,E1 20837.436,E2 20837.436} C_VEL
LIN {X 0,Y 441.199,Z 523.842,A -85,B 0,C 180,E1 20833.703,E2 20833.703} C_VEL
LIN {X 0,Y 441.195,Z 523.837,A -85,B 0,C 180,E1 20829.89,E2 20829.89} C_VEL
LIN {X 0,Y 441.264,Z 524.242,A -85,B 0,C 180,E1 20829.45,E2 20829.45} C_VEL
LIN {X 0,Y 449.763,Z 548.089,A -85,B 0,C 180,E1 20826.198,E2 20826.198} C_VEL
LIN {X 0,Y 454.302,Z 561.611,A -85,B 0,C 180,E1 20824.498,E2 20824.498} C_VEL
LIN {X 0,Y 450.678,Z 607.406,A -85,B 0,C 180,E1 20820.312,E2 20820.312} C_VEL
LIN {X 0,Y 450.091,Z 616.564,A -85,B 0,C 180,E1 20819.515,E2 20819.515} C_VEL
LIN {X 0,Y 452.509,Z 638.088,A -85,B 0,C 180,E1 20819.009,E2 20819.009} C_VEL
LIN {X 0,Y 450.148,Z 818.07,A -85,B 0,C 180,E1 20816.117,E2 20816.117} C_VEL
LIN {X 0,Y 449.384,Z 836.894,A -85,B 0,C 180,E1 20815.588,E2 20815.588} C_VEL
LIN {X 0,Y 448.385,Z 854.799,A -85,B 0,C 180,E1 20814.855,E2 20814.855} C_VEL
LIN {X 0,Y 447.257,Z 872.404,A -85,B 0,C 180,E1 20813.889,E2 20813.889} C_VEL
LIN {X 0,Y 445.974,Z 889.609,A -85,B 0,C 180,E1 20812.682,E2 20812.682} C_VEL
LIN {X 0,Y 444.725,Z 905.61,A -85,B 0,C 180,E1 20811.29,E2 20811.29} C_VEL
LIN {X 0,Y 443.55,Z 920.683,A -85,B 0,C 180,E1 20809.694,E2 20809.694} C_VEL
LIN {X 0,Y 442.469,Z 934.74,A -85,B 0,C 180,E1 20807.898,E2 20807.898} C_VEL
LIN {X 0,Y 441.588,Z 947.671,A -85,B 0,C 180,E1 20805.901,E2 20805.901} C_VEL
LIN {X 0,Y 440.936,Z 958.989,A -85,B 0,C 180,E1 20803.775,E2 20803.775} C_VEL
LIN {X 0,Y 440.531,Z 968.673,A -85,B 0,C 180,E1 20801.522,E2 20801.522} C_VEL
LIN {X 0,Y 440.344,Z 976.325,A -85,B 0,C 180,E1 20799.278,E2 20799.278} C_VEL
LIN {X 0,Y 440.287,Z 982.167,A -85,B 0,C 180,E1 20797.045,E2 20797.045} C_VEL
LIN {X 0,Y 440.329,Z 986.512,A -85,B 0,C 180,E1 20794.69,E2 20794.69} C_VEL
LIN {X 0,Y 440.393,Z 989.079,A -85,B 0,C 180,E1 20792.344,E2 20792.344} C_VEL
LIN {X 0,Y 440.43,Z 989.917,A -85,B 0,C 180,E1 20790.002,E2 20790.002} C_VEL
LIN {X 0,Y 440.401,Z 989.033,A -85,B 0,C 180,E1 20787.66,E2 20787.66} C_VEL
LIN {X 0,Y 440.341,Z 986.42,A -85,B 0,C 180,E1 20785.313,E2 20785.313} C_VEL
LIN {X 0,Y 440.301,Z 982.031,A -85,B 0,C 180,E1 20782.959,E2 20782.959} C_VEL
LIN {X 0,Y 440.364,Z 975.765,A -85,B 0,C 180,E1 20780.594,E2 20780.594} C_VEL
LIN {X 0,Y 440.556,Z 967.956,A -85,B 0,C 180,E1 20778.349,E2 20778.349} C_VEL
LIN {X 0,Y 440.972,Z 958.074,A -85,B 0,C 180,E1 20776.096,E2 20776.096} C_VEL
LIN {X 0,Y 441.584,Z 947.391,A -85,B 0,C 180,E1 20774.102,E2 20774.102} C_VEL
LIN {X 0,Y 442.456,Z 934.435,A -85,B 0,C 180,E1 20772.105,E2 20772.105} C_VEL
LIN {X 0,Y 443.528,Z 920.363,A -85,B 0,C 180,E1 20770.308,E2 20770.308} C_VEL
LIN {X 0,Y 444.697,Z 905.29,A -85,B 0,C 180,E1 20768.712,E2 20768.712} C_VEL
LIN {X 0,Y 446.017,Z 888.511,A -85,B 0,C 180,E1 20767.254,E2 20767.254} C_VEL
LIN {X 0,Y 447.284,Z 871.637,A -85,B 0,C 180,E1 20766.074,E2 20766.074} C_VEL
LIN {X 0,Y 448.416,Z 854.283,A -85,B 0,C 180,E1 20765.118,E2 20765.118} C_VEL
LIN {X 0,Y 449.457,Z 836.1,A -85,B 0,C 180,E1 20764.371,E2 20764.371} C_VEL
LIN {X 0,Y 450.244,Z 817.144,A -85,B 0,C 180,E1 20763.84,E2 20763.84} C_VEL
LIN {X 0,Y 452.564,Z 635.219,A -85,B 0,C 180,E1 20760.877,E2 20760.877} C_VEL
LIN {X 0,Y 450.327,Z 616.549,A -85,B 0,C 180,E1 20760.397,E2 20760.397} C_VEL
LIN {X 0,Y 453.86,Z 573.645,A -85,B 0,C 180,E1 20756.435,E2 20756.435} C_VEL
LIN {X 0,Y 454.794,Z 561.884,A -85,B 0,C 180,E1 20755.296,E2 20755.296} C_VEL
LIN {X 0,Y 448.552,Z 543.2,A -85,B 0,C 180,E1 20752.729,E2 20752.729} C_VEL
LIN {X 0,Y 442.319,Z 527.058,A -85,B 0,C 180,E1 20750.225,E2 20750.225} C_VEL
LIN {X 0,Y 441.182,Z 523.99,A -85,B 0,C 180,E1 20749.645,E2 20749.645} C_VEL
LIN {X 0,Y 441.192,Z 523.841,A -85,B 0,C 180,E1 20746.101,E2 20746.101} C_VEL
LIN {X 0,Y 441.194,Z 523.836,A -85,B 0,C 180,E1 20742.305,E2 20742.305} C_VEL
LIN {X 0,Y 441.155,Z 523.835,A -85,B 0,C 180,E1 20738.722,E2 20738.722} C_VEL
LIN {X 0,Y 441.142,Z 523.84,A -85,B 0,C 180,E1 20734.99,E2 20734.99} C_VEL
LIN {X 0,Y 441.148,Z 523.839,A -85,B 0,C 180,E1 20731.267,E2 20731.267} C_VEL
LIN {X 0,Y 441.183,Z 523.831,A -85,B 0,C 180,E1 20727.684,E2 20727.684} C_VEL
LIN {X 0,Y 441.17,Z 523.831,A -85,B 0,C 180,E1 20723.934,E2 20723.934} C_VEL
LIN {X 0,Y 441.128,Z 523.844,A -85,B 0,C 180,E1 20720.429,E2 20720.429} C_VEL
LIN {X 0,Y 441.125,Z 523.847,A -85,B 0,C 180,E1 20716.73,E2 20716.73} C_VEL
LIN {X 0,Y 441.148,Z 523.841,A -85,B 0,C 180,E1 20713.1,E2 20713.1} C_VEL
LIN {X 0,Y 441.167,Z 523.829,A -85,B 0,C 180,E1 20709.391,E2 20709.391} C_VEL
LIN {X 0,Y 441.129,Z 523.845,A -85,B 0,C 180,E1 20705.854,E2 20705.854} C_VEL
LIN {X 0,Y 441.125,Z 523.846,A -85,B 0,C 180,E1 20702.208,E2 20702.208} C_VEL
LIN {X 0,Y 441.15,Z 523.841,A -85,B 0,C 180,E1 20698.571,E2 20698.571} C_VEL
LIN {X 0,Y 441.184,Z 523.828,A -85,B 0,C 180,E1 20694.929,E2 20694.929} C_VEL
LIN {X 0,Y 441.159,Z 523.836,A -85,B 0,C 180,E1 20691.265,E2 20691.265} C_VEL
LIN {X 0,Y 441.144,Z 523.845,A -85,B 0,C 180,E1 20687.565,E2 20687.565} C_VEL
LIN {X 0,Y 441.148,Z 523.844,A -85,B 0,C 180,E1 20683.812,E2 20683.812} C_VEL
LIN {X 0,Y 441.173,Z 523.84,A -85,B 0,C 180,E1 20680.124,E2 20680.124} C_VEL
LIN {X 0,Y 441.202,Z 523.834,A -85,B 0,C 180,E1 20676.493,E2 20676.493} C_VEL
LIN {X 0,Y 441.178,Z 523.836,A -85,B 0,C 180,E1 20672.754,E2 20672.754} C_VEL
LIN {X 0,Y 441.165,Z 523.847,A -85,B 0,C 180,E1 20669.037,E2 20669.037} C_VEL
LIN {X 0,Y 441.23,Z 524.102,A -85,B 0,C 180,E1 20665.891,E2 20665.891} C_VEL
LIN {X 0,Y 446.318,Z 539.752,A -85,B 0,C 180,E1 20662.78,E2 20662.78} C_VEL
LIN {X 0,Y 450.592,Z 555.435,A -85,B 0,C 180,E1 20659.946,E2 20659.946} C_VEL
LIN {X 0,Y 450.746,Z 558.071,A -85,B 0,C 180,E1 20659.531,E2 20659.531} C_VEL
LIN {X 0,Y 448.339,Z 586.159,A -85,B 0,C 180,E1 20655.551,E2 20655.551} C_VEL
LIN {X 0,Y 446.225,Z 615.033,A -85,B 0,C 180,E1 20651.542,E2 20651.542} C_VEL
LIN {X 0,Y 445.253,Z 631.171,A -85,B 0,C 180,E1 20649.371,E2 20649.371} C_VEL
LIN {X 0,Y 449.009,Z 652.208,A -85,B 0,C 180,E1 20648.73,E2 20648.73} C_VEL
LIN {X 0,Y 447.387,Z 751.408,A -85,B 0,C 180,E1 20646.994,E2 20646.994} C_VEL
LIN {X 0,Y 446.976,Z 767.48,A -85,B 0,C 180,E1 20646.461,E2 20646.461} C_VEL
LIN {X 0,Y 446.346,Z 782.167,A -85,B 0,C 180,E1 20645.717,E2 20645.717} C_VEL
LIN {X 0,Y 445.578,Z 795.727,A -85,B 0,C 180,E1 20644.785,E2 20644.785} C_VEL
LIN {X 0,Y 444.641,Z 808.936,A -85,B 0,C 180,E1 20643.591,E2 20643.591} C_VEL
LIN {X 0,Y 443.268,Z 814.996,A -85,B 0,C 180,E1 20642.988,E2 20642.988} C_VEL
LIN {X 0,Y 438.213,Z 825.48,A -85,B 0,C 180,E1 20641.853,E2 20641.853} C_VEL
LIN {X 0,Y 435.62,Z 831.404,A -85,B 0,C 180,E1 20641.046,E2 20641.046} C_VEL
LIN {X 0,Y 435.041,Z 834.089,A -85,B 0,C 180,E1 20640.594,E2 20640.594} C_VEL
LIN {X 0,Y 434.293,Z 842.348,A -85,B 0,C 180,E1 20638.908,E2 20638.908} C_VEL
LIN {X 0,Y 433.685,Z 849.398,A -85,B 0,C 180,E1 20637.008,E2 20637.008} C_VEL
LIN {X 0,Y 433.281,Z 854.404,A -85,B 0,C 180,E1 20635.122,E2 20635.122} C_VEL
LIN {X 0,Y 433.021,Z 857.905,A -85,B 0,C 180,E1 20633.108,E2 20633.108} C_VEL
LIN {X 0,Y 432.878,Z 859.624,A -85,B 0,C 180,E1 20630.975,E2 20630.975} C_VEL
LIN {X 0,Y 432.854,Z 859.525,A -85,B 0,C 180,E1 20629.004,E2 20629.004} C_VEL
LIN {X 0,Y 432.944,Z 857.641,A -85,B 0,C 180,E1 20626.914,E2 20626.914} C_VEL
LIN {X 0,Y 433.163,Z 853.835,A -85,B 0,C 180,E1 20624.843,E2 20624.843} C_VEL
LIN {X 0,Y 433.516,Z 848.478,A -85,B 0,C 180,E1 20622.925,E2 20622.925} C_VEL
LIN {X 0,Y 434.065,Z 841.112,A -85,B 0,C 180,E1 20621.02,E2 20621.02} C_VEL
LIN {X 0,Y 434.78,Z 832.074,A -85,B 0,C 180,E1 20619.261,E2 20619.261} C_VEL
LIN {X 0,Y 435.588,Z 821.902,A -85,B 0,C 180,E1 20617.715,E2 20617.715} C_VEL
LIN {X 0,Y 436.461,Z 810.162,A -85,B 0,C 180,E1 20616.311,E2 20616.311} C_VEL
LIN {X 0,Y 437.342,Z 797.261,A -85,B 0,C 180,E1 20615.113,E2 20615.113} C_VEL
LIN {X 0,Y 438.103,Z 784.189,A -85,B 0,C 180,E1 20614.172,E2 20614.172} C_VEL
LIN {X 0,Y 438.778,Z 768.778,A -85,B 0,C 180,E1 20613.362,E2 20613.362} C_VEL
LIN {X 0,Y 439.201,Z 753.496,A -85,B 0,C 180,E1 20612.828,E2 20612.828} C_VEL
LIN {X 0,Y 439.626,Z 724.724,A -85,B 0,C 180,E1 20612.277,E2 20612.277} C_VEL
LIN {X 0,Y 440.521,Z 650.734,A -85,B 0,C 180,E1 20611.01,E2 20611.01} C_VEL
LIN {X 0,Y 437.037,Z 631.092,A -85,B 0,C 180,E1 20610.457,E2 20610.457} C_VEL
LIN {X 0,Y 438.815,Z 601.826,A -85,B 0,C 180,E1 20606.472,E2 20606.472} C_VEL
LIN {X 0,Y 440.864,Z 573.767,A -85,B 0,C 180,E1 20602.571,E2 20602.571} C_VEL
LIN {X 0,Y 442.096,Z 556.35,A -85,B 0,C 180,E1 20600.102,E2 20600.102} C_VEL
LIN {X 0,Y 437.047,Z 537.785,A -85,B 0,C 180,E1 20596.909,E2 20596.909} C_VEL
LIN {X 0,Y 433.197,Z 524.943,A -85,B 0,C 180,E1 20594.539,E2 20594.539} C_VEL
LIN {X 0,Y 433.202,Z 524.831,A -85,B 0,C 180,E1 20590.868,E2 20590.868} C_VEL
LIN {X 0,Y 433.238,Z 524.798,A -85,B 0,C 180,E1 20587.187,E2 20587.187} C_VEL
LIN {X 0,Y 433.223,Z 524.834,A -85,B 0,C 180,E1 20583.276,E2 20583.276} C_VEL
LIN {X 0,Y 433.179,Z 524.791,A -85,B 0,C 180,E1 20579.637,E2 20579.637} C_VEL
LIN {X 0,Y 433.178,Z 524.836,A -85,B 0,C 180,E1 20575.884,E2 20575.884} C_VEL
LIN {X 0,Y 433.187,Z 524.829,A -85,B 0,C 180,E1 20572.125,E2 20572.125} C_VEL
LIN {X 0,Y 433.233,Z 524.821,A -85,B 0,C 180,E1 20568.522,E2 20568.522} C_VEL
LIN {X 0,Y 433.226,Z 524.834,A -85,B 0,C 180,E1 20564.699,E2 20564.699} C_VEL
LIN {X 0,Y 433.192,Z 524.816,A -85,B 0,C 180,E1 20560.999,E2 20560.999} C_VEL
LIN {X 0,Y 433.186,Z 524.835,A -85,B 0,C 180,E1 20557.376,E2 20557.376} C_VEL
LIN {X 0,Y 433.201,Z 524.814,A -85,B 0,C 180,E1 20553.638,E2 20553.638} C_VEL
LIN {X 0,Y 433.235,Z 524.832,A -85,B 0,C 180,E1 20549.901,E2 20549.901} C_VEL
LIN {X 0,Y 433.235,Z 524.806,A -85,B 0,C 180,E1 20546.14,E2 20546.14} C_VEL
LIN {X 0,Y 433.201,Z 524.832,A -85,B 0,C 180,E1 20542.529,E2 20542.529} C_VEL
LIN {X 0,Y 433.195,Z 524.818,A -85,B 0,C 180,E1 20538.853,E2 20538.853} C_VEL
LIN {X 0,Y 433.211,Z 524.828,A -85,B 0,C 180,E1 20535.118,E2 20535.118} C_VEL
LIN {X 0,Y 433.246,Z 524.821,A -85,B 0,C 180,E1 20531.448,E2 20531.448} C_VEL
LIN {X 0,Y 433.231,Z 524.806,A -85,B 0,C 180,E1 20527.693,E2 20527.693} C_VEL
LIN {X 0,Y 433.209,Z 524.832,A -85,B 0,C 180,E1 20523.971,E2 20523.971} C_VEL
LIN {X 0,Y 433.2,Z 524.803,A -85,B 0,C 180,E1 20520.265,E2 20520.265} C_VEL
LIN {X 0,Y 433.223,Z 524.831,A -85,B 0,C 180,E1 20516.56,E2 20516.56} C_VEL
LIN {X 0,Y 433.257,Z 524.805,A -85,B 0,C 180,E1 20512.841,E2 20512.841} C_VEL
LIN {X 0,Y 433.251,Z 524.833,A -85,B 0,C 180,E1 20508.957,E2 20508.957} C_VEL
LIN {X 0,Y 433.223,Z 524.814,A -85,B 0,C 180,E1 20505.234,E2 20505.234} C_VEL
LIN {X 0,Y 433.213,Z 524.833,A -85,B 0,C 180,E1 20501.538,E2 20501.538} C_VEL
LIN {X 0,Y 433.217,Z 524.825,A -85,B 0,C 180,E1 20497.736,E2 20497.736} C_VEL
LIN {X 0,Y 433.251,Z 524.816,A -85,B 0,C 180,E1 20494.14,E2 20494.14} C_VEL
LIN {X 0,Y 433.262,Z 524.828,A -85,B 0,C 180,E1 20490.406,E2 20490.406} C_VEL
LIN {X 0,Y 433.234,Z 524.832,A -85,B 0,C 180,E1 20486.659,E2 20486.659} C_VEL
LIN {X 0,Y 433.221,Z 524.832,A -85,B 0,C 180,E1 20482.96,E2 20482.96} C_VEL
LIN {X 0,Y 433.228,Z 524.832,A -85,B 0,C 180,E1 20479.197,E2 20479.197} C_VEL
LIN {X 0,Y 433.249,Z 524.823,A -85,B 0,C 180,E1 20475.447,E2 20475.447} C_VEL
LIN {X 0,Y 433.264,Z 524.831,A -85,B 0,C 180,E1 20471.608,E2 20471.608} C_VEL
LIN {X 0,Y 433.271,Z 525.043,A -85,B 0,C 180,E1 20470.124,E2 20470.124} C_VEL
LIN {X 0,Y 436.371,Z 533.732,A -85,B 0,C 180,E1 20468.827,E2 20468.827} C_VEL
LIN {X 0,Y 444.185,Z 555.939,A -85,B 0,C 180,E1 20465.82,E2 20465.82} C_VEL
LIN {X 0,Y 446.898,Z 564.091,A -85,B 0,C 180,E1 20464.785,E2 20464.785} C_VEL
LIN {X 0,Y 443.302,Z 607.369,A -85,B 0,C 180,E1 20460.758,E2 20460.758} C_VEL
LIN {X 0,Y 442.66,Z 616.905,A -85,B 0,C 180,E1 20459.918,E2 20459.918} C_VEL
LIN {X 0,Y 445.125,Z 639.034,A -85,B 0,C 180,E1 20459.393,E2 20459.393} C_VEL
LIN {X 0,Y 442.637,Z 817.576,A -85,B 0,C 180,E1 20456.477,E2 20456.477} C_VEL
LIN {X 0,Y 441.836,Z 836.312,A -85,B 0,C 180,E1 20455.942,E2 20455.942} C_VEL
LIN {X 0,Y 440.783,Z 854.24,A -85,B 0,C 180,E1 20455.195,E2 20455.195} C_VEL
LIN {X 0,Y 439.59,Z 871.935,A -85,B 0,C 180,E1 20454.205,E2 20454.205} C_VEL
LIN {X 0,Y 438.233,Z 889.308,A -85,B 0,C 180,E1 20452.963,E2 20452.963} C_VEL
LIN {X 0,Y 436.918,Z 905.25,A -85,B 0,C 180,E1 20451.549,E2 20451.549} C_VEL
LIN {X 0,Y 435.69,Z 920.253,A -85,B 0,C 180,E1 20449.925,E2 20449.925} C_VEL
LIN {X 0,Y 434.559,Z 934.215,A -85,B 0,C 180,E1 20448.096,E2 20448.096} C_VEL
LIN {X 0,Y 433.638,Z 947.06,A -85,B 0,C 180,E1 20446.063,E2 20446.063} C_VEL
LIN {X 0,Y 432.965,Z 958.272,A -85,B 0,C 180,E1 20443.897,E2 20443.897} C_VEL
LIN {X 0,Y 432.553,Z 967.872,A -85,B 0,C 180,E1 20441.602,E2 20441.602} C_VEL
LIN {X 0,Y 432.379,Z 975.453,A -85,B 0,C 180,E1 20439.316,E2 20439.316} C_VEL
LIN {X 0,Y 432.34,Z 981.222,A -85,B 0,C 180,E1 20437.042,E2 20437.042} C_VEL
LIN {X 0,Y 432.398,Z 985.406,A -85,B 0,C 180,E1 20434.708,E2 20434.708} C_VEL
LIN {X 0,Y 432.472,Z 987.897,A -85,B 0,C 180,E1 20432.386,E2 20432.386} C_VEL
LIN {X 0,Y 432.517,Z 988.738,A -85,B 0,C 180,E1 20430.002,E2 20430.002} C_VEL
LIN {X 0,Y 432.48,Z 987.848,A -85,B 0,C 180,E1 20427.617,E2 20427.617} C_VEL
LIN {X 0,Y 432.405,Z 985.223,A -85,B 0,C 180,E1 20425.227,E2 20425.227} C_VEL
LIN {X 0,Y 432.351,Z 980.75,A -85,B 0,C 180,E1 20422.797,E2 20422.797} C_VEL
LIN {X 0,Y 432.399,Z 974.517,A -85,B 0,C 180,E1 20420.419,E2 20420.419} C_VEL
LIN {X 0,Y 432.595,Z 966.671,A -85,B 0,C 180,E1 20418.132,E2 20418.132} C_VEL
LIN {X 0,Y 433.037,Z 956.739,A -85,B 0,C 180,E1 20415.836,E2 20415.836} C_VEL
LIN {X 0,Y 433.684,Z 946.002,A -85,B 0,C 180,E1 20413.805,E2 20413.805} C_VEL
LIN {X 0,Y 434.581,Z 933.496,A -85,B 0,C 180,E1 20411.843,E2 20411.843} C_VEL
LIN {X 0,Y 435.717,Z 919.458,A -85,B 0,C 180,E1 20410.01,E2 20410.01} C_VEL
LIN {X 0,Y 436.956,Z 904.465,A -85,B 0,C 180,E1 20408.386,E2 20408.386} C_VEL
LIN {X 0,Y 438.368,Z 887.736,A -85,B 0,C 180,E1 20406.906,E2 20406.906} C_VEL
LIN {X 0,Y 439.716,Z 870.79,A -85,B 0,C 180,E1 20405.7,E2 20405.7} C_VEL
LIN {X 0,Y 440.916,Z 853.504,A -85,B 0,C 180,E1 20404.734,E2 20404.734} C_VEL
LIN {X 0,Y 442.008,Z 835.421,A -85,B 0,C 180,E1 20403.979,E2 20403.979} C_VEL
LIN {X 0,Y 442.836,Z 816.609,A -85,B 0,C 180,E1 20403.444,E2 20403.444} C_VEL
LIN {X 0,Y 445.3,Z 636.117,A -85,B 0,C 180,E1 20400.454,E2 20400.454} C_VEL
LIN {X 0,Y 443.018,Z 616.396,A -85,B 0,C 180,E1 20399.917,E2 20399.917} C_VEL
LIN {X 0,Y 446.915,Z 573.377,A -85,B 0,C 180,E1 20395.842,E2 20395.842} C_VEL
LIN {X 0,Y 447.731,Z 565.133,A -85,B 0,C 180,E1 20395.042,E2 20395.042} C_VEL
LIN {X 0,Y 441.738,Z 547.049,A -85,B 0,C 180,E1 20392.498,E2 20392.498} C_VEL
LIN {X 0,Y 435.775,Z 531.457,A -85,B 0,C 180,E1 20390.026,E2 20390.026} C_VEL
LIN {X 0,Y 433.262,Z 525.021,A -85,B 0,C 180,E1 20388.876,E2 20388.876} C_VEL
LIN {X 0,Y 433.217,Z 524.832,A -85,B 0,C 180,E1 20385.117,E2 20385.117} C_VEL
LIN {X 0,Y 433.212,Z 524.829,A -85,B 0,C 180,E1 20381.307,E2 20381.307} C_VEL
LIN {X 0,Y 433.231,Z 524.832,A -85,B 0,C 180,E1 20377.673,E2 20377.673} C_VEL
LIN {X 0,Y 433.254,Z 524.831,A -85,B 0,C 180,E1 20373.951,E2 20373.951} C_VEL
LIN {X 0,Y 433.231,Z 524.831,A -85,B 0,C 180,E1 20370.207,E2 20370.207} C_VEL
LIN {X 0,Y 433.197,Z 524.833,A -85,B 0,C 180,E1 20366.6,E2 20366.6} C_VEL
LIN {X 0,Y 433.192,Z 524.83,A -85,B 0,C 180,E1 20362.815,E2 20362.815} C_VEL
LIN {X 0,Y 433.205,Z 524.82,A -85,B 0,C 180,E1 20359.132,E2 20359.132} C_VEL
LIN {X 0,Y 433.235,Z 524.819,A -85,B 0,C 180,E1 20355.391,E2 20355.391} C_VEL
LIN {X 0,Y 433.22,Z 524.836,A -85,B 0,C 180,E1 20351.583,E2 20351.583} C_VEL
LIN {X 0,Y 433.192,Z 524.832,A -85,B 0,C 180,E1 20347.827,E2 20347.827} C_VEL
LIN {X 0,Y 433.182,Z 524.822,A -85,B 0,C 180,E1 20344.103,E2 20344.103} C_VEL
LIN {X 0,Y 433.19,Z 524.822,A -85,B 0,C 180,E1 20340.264,E2 20340.264} C_VEL
LIN {X 0,Y 433.215,Z 524.829,A -85,B 0,C 180,E1 20336.559,E2 20336.559} C_VEL
LIN {X 0,Y 433.259,Z 524.832,A -85,B 0,C 180,E1 20332.841,E2 20332.841} C_VEL
LIN {X 0,Y 433.243,Z 524.829,A -85,B 0,C 180,E1 20328.956,E2 20328.956} C_VEL
LIN {X 0,Y 433.219,Z 524.828,A -85,B 0,C 180,E1 20325.224,E2 20325.224} C_VEL
LIN {X 0,Y 433.21,Z 524.83,A -85,B 0,C 180,E1 20321.529,E2 20321.529} C_VEL
LIN {X 0,Y 433.218,Z 524.834,A -85,B 0,C 180,E1 20317.727,E2 20317.727} C_VEL
LIN {X 0,Y 433.243,Z 524.831,A -85,B 0,C 180,E1 20313.992,E2 20313.992} C_VEL
LIN {X 0,Y 433.267,Z 524.822,A -85,B 0,C 180,E1 20310.181,E2 20310.181} C_VEL
LIN {X 0,Y 433.283,Z 525.114,A -85,B 0,C 180,E1 20306.651,E2 20306.651} C_VEL
LIN {X 0,Y 438.059,Z 539.599,A -85,B 0,C 180,E1 20303.67,E2 20303.67} C_VEL
LIN {X 0,Y 442.085,Z 553.467,A -85,B 0,C 180,E1 20301.042,E2 20301.042} C_VEL
LIN {X 0,Y 443.531,Z 559.685,A -85,B 0,C 180,E1 20299.938,E2 20299.938} C_VEL
LIN {X 0,Y 440.978,Z 587.428,A -85,B 0,C 180,E1 20295.944,E2 20295.944} C_VEL
LIN {X 0,Y 438.723,Z 616.188,A -85,B 0,C 180,E1 20291.887,E2 20291.887} C_VEL
LIN {X 0,Y 437.765,Z 630.839,A -85,B 0,C 180,E1 20289.876,E2 20289.876} C_VEL
LIN {X 0,Y 441.797,Z 653.011,A -85,B 0,C 180,E1 20289.167,E2 20289.167} C_VEL
LIN {X 0,Y 440.053,Z 752.018,A -85,B 0,C 180,E1 20287.399,E2 20287.399} C_VEL
LIN {X 0,Y 439.605,Z 768.275,A -85,B 0,C 180,E1 20286.849,E2 20286.849} C_VEL
LIN {X 0,Y 438.95,Z 782.584,A -85,B 0,C 180,E1 20286.115,E2 20286.115} C_VEL
LIN {X 0,Y 438.141,Z 796.107,A -85,B 0,C 180,E1 20285.179,E2 20285.179} C_VEL
LIN {X 0,Y 437.139,Z 809.36,A -85,B 0,C 180,E1 20283.973,E2 20283.973} C_VEL
LIN {X 0,Y 436.236,Z 820.609,A -85,B 0,C 180,E1 20282.663,E2 20282.663} C_VEL
LIN {X 0,Y 435.273,Z 831.569,A -85,B 0,C 180,E1 20281.039,E2 20281.039} C_VEL
LIN {X 0,Y 435.041,Z 834.089,A -85,B 0,C 180,E1 20280.594,E2 20280.594} C_VEL
LIN {X 0,Y 433.684,Z 838.644,A -85,B 0,C 180,E1 20279.783,E2 20279.783} C_VEL
LIN {X 0,Y 428.714,Z 846.279,A -85,B 0,C 180,E1 20278.275,E2 20278.275} C_VEL
LIN {X 0,Y 426.235,Z 850.257,A -85,B 0,C 180,E1 20277.259,E2 20277.259} C_VEL
LIN {X 0,Y 425.738,Z 851.957,A -85,B 0,C 180,E1 20276.712,E2 20276.712} C_VEL
LIN {X 0,Y 425.333,Z 856.676,A -85,B 0,C 180,E1 20274.732,E2 20274.732} C_VEL
LIN {X 0,Y 425.065,Z 859.813,A -85,B 0,C 180,E1 20272.542,E2 20272.542} C_VEL
LIN {X 0,Y 424.953,Z 860.931,A -85,B 0,C 180,E1 20270.519,E2 20270.519} C_VEL
LIN {X 0,Y 424.96,Z 860.353,A -85,B 0,C 180,E1 20268.374,E2 20268.374} C_VEL
LIN {X 0,Y 425.09,Z 857.888,A -85,B 0,C 180,E1 20266.251,E2 20266.251} C_VEL
LIN {X 0,Y 425.35,Z 853.893,A -85,B 0,C 180,E1 20264.286,E2 20264.286} C_VEL
LIN {X 0,Y 425.814,Z 847.607,A -85,B 0,C 180,E1 20262.198,E2 20262.198} C_VEL
LIN {X 0,Y 426.471,Z 839.53,A -85,B 0,C 180,E1 20260.261,E2 20260.261} C_VEL
LIN {X 0,Y 427.233,Z 830.583,A -85,B 0,C 180,E1 20258.612,E2 20258.612} C_VEL
LIN {X 0,Y 428.156,Z 819.618,A -85,B 0,C 180,E1 20257.023,E2 20257.023} C_VEL
LIN {X 0,Y 429.108,Z 807.096,A -85,B 0,C 180,E1 20255.614,E2 20255.614} C_VEL
LIN {X 0,Y 429.975,Z 794.811,A -85,B 0,C 180,E1 20254.533,E2 20254.533} C_VEL
LIN {X 0,Y 430.822,Z 779.866,A -85,B 0,C 180,E1 20253.531,E2 20253.531} C_VEL
LIN {X 0,Y 431.454,Z 764.143,A -85,B 0,C 180,E1 20252.791,E2 20252.791} C_VEL
LIN {X 0,Y 431.815,Z 748.853,A -85,B 0,C 180,E1 20252.333,E2 20252.333} C_VEL
LIN {X 0,Y 433.139,Z 651.892,A -85,B 0,C 180,E1 20250.623,E2 20250.623} C_VEL
LIN {X 0,Y 429.415,Z 630.638,A -85,B 0,C 180,E1 20249.998,E2 20249.998} C_VEL
LIN {X 0,Y 431.394,Z 600.946,A -85,B 0,C 180,E1 20245.878,E2 20245.878} C_VEL
LIN {X 0,Y 433.563,Z 572.859,A -85,B 0,C 180,E1 20241.912,E2 20241.912} C_VEL
LIN {X 0,Y 434.642,Z 559.009,A -85,B 0,C 180,E1 20239.928,E2 20239.928} C_VEL
LIN {X 0,Y 429.863,Z 541.257,A -85,B 0,C 180,E1 20236.823,E2 20236.823} C_VEL
LIN {X 0,Y 425.274,Z 525.95,A -85,B 0,C 180,E1 20233.963,E2 20233.963} C_VEL
LIN {X 0,Y 425.245,Z 525.82,A -85,B 0,C 180,E1 20230.21,E2 20230.21} C_VEL
LIN {X 0,Y 425.24,Z 525.786,A -85,B 0,C 180,E1 20226.44,E2 20226.44} C_VEL
LIN {X 0,Y 425.266,Z 525.823,A -85,B 0,C 180,E1 20222.712,E2 20222.712} C_VEL
LIN {X 0,Y 425.29,Z 525.773,A -85,B 0,C 180,E1 20219.012,E2 20219.012} C_VEL
LIN {X 0,Y 425.258,Z 525.825,A -85,B 0,C 180,E1 20215.322,E2 20215.322} C_VEL
LIN {X 0,Y 425.241,Z 525.819,A -85,B 0,C 180,E1 20211.632,E2 20211.632} C_VEL
LIN {X 0,Y 425.241,Z 525.81,A -85,B 0,C 180,E1 20207.745,E2 20207.745} C_VEL
LIN {X 0,Y 425.259,Z 525.823,A -85,B 0,C 180,E1 20203.993,E2 20203.993} C_VEL
LIN {X 0,Y 425.297,Z 525.804,A -85,B 0,C 180,E1 20200.28,E2 20200.28} C_VEL
LIN {X 0,Y 425.287,Z 525.819,A -85,B 0,C 180,E1 20196.485,E2 20196.485} C_VEL
LIN {X 0,Y 425.265,Z 525.806,A -85,B 0,C 180,E1 20192.684,E2 20192.684} C_VEL
LIN {X 0,Y 425.251,Z 525.822,A -85,B 0,C 180,E1 20188.97,E2 20188.97} C_VEL
LIN {X 0,Y 425.256,Z 525.805,A -85,B 0,C 180,E1 20185.155,E2 20185.155} C_VEL
LIN {X 0,Y 425.281,Z 525.82,A -85,B 0,C 180,E1 20181.414,E2 20181.414} C_VEL
LIN {X 0,Y 425.306,Z 525.79,A -85,B 0,C 180,E1 20177.654,E2 20177.654} C_VEL
LIN {X 0,Y 425.295,Z 525.819,A -85,B 0,C 180,E1 20173.857,E2 20173.857} C_VEL
LIN {X 0,Y 425.265,Z 525.805,A -85,B 0,C 180,E1 20170.157,E2 20170.157} C_VEL
LIN {X 0,Y 425.261,Z 525.814,A -85,B 0,C 180,E1 20166.345,E2 20166.345} C_VEL
LIN {X 0,Y 425.27,Z 525.812,A -85,B 0,C 180,E1 20162.561,E2 20162.561} C_VEL
LIN {X 0,Y 425.305,Z 525.802,A -85,B 0,C 180,E1 20158.923,E2 20158.923} C_VEL
LIN {X 0,Y 425.309,Z 525.816,A -85,B 0,C 180,E1 20155.145,E2 20155.145} C_VEL
LIN {X 0,Y 425.278,Z 525.8,A -85,B 0,C 180,E1 20151.482,E2 20151.482} C_VEL
LIN {X 0,Y 425.27,Z 525.821,A -85,B 0,C 180,E1 20147.784,E2 20147.784} C_VEL
LIN {X 0,Y 425.281,Z 525.812,A -85,B 0,C 180,E1 20144.034,E2 20144.034} C_VEL
LIN {X 0,Y 425.311,Z 525.809,A -85,B 0,C 180,E1 20140.356,E2 20140.356} C_VEL
LIN {X 0,Y 425.32,Z 525.818,A -85,B 0,C 180,E1 20136.591,E2 20136.591} C_VEL
LIN {X 0,Y 425.302,Z 525.807,A -85,B 0,C 180,E1 20132.698,E2 20132.698} C_VEL
LIN {X 0,Y 425.281,Z 525.813,A -85,B 0,C 180,E1 20129.011,E2 20129.011} C_VEL
LIN {X 0,Y 425.278,Z 525.816,A -85,B 0,C 180,E1 20125.133,E2 20125.133} C_VEL
LIN {X 0,Y 425.289,Z 525.813,A -85,B 0,C 180,E1 20121.291,E2 20121.291} C_VEL
LIN {X 0,Y 425.311,Z 525.813,A -85,B 0,C 180,E1 20117.569,E2 20117.569} C_VEL
LIN {X 0,Y 425.321,Z 525.821,A -85,B 0,C 180,E1 20113.718,E2 20113.718} C_VEL
LIN {X 0,Y 425.323,Z 526.083,A -85,B 0,C 180,E1 20110.739,E2 20110.739} C_VEL
LIN {X 0,Y 432.811,Z 546.893,A -85,B 0,C 180,E1 20107.7,E2 20107.7} C_VEL
LIN {X 0,Y 439.549,Z 566.785,A -85,B 0,C 180,E1 20105.054,E2 20105.054} C_VEL
LIN {X 0,Y 435.494,Z 612.597,A -85,B 0,C 180,E1 20100.719,E2 20100.719} C_VEL
LIN {X 0,Y 435.248,Z 617.157,A -85,B 0,C 180,E1 20100.34,E2 20100.34} C_VEL
LIN {X 0,Y 437.76,Z 639.987,A -85,B 0,C 180,E1 20099.788,E2 20099.788} C_VEL
LIN {X 0,Y 435.148,Z 816.942,A -85,B 0,C 180,E1 20096.853,E2 20096.853} C_VEL
LIN {X 0,Y 434.312,Z 835.619,A -85,B 0,C 180,E1 20096.311,E2 20096.311} C_VEL
LIN {X 0,Y 433.185,Z 853.921,A -85,B 0,C 180,E1 20095.533,E2 20095.533} C_VEL
LIN {X 0,Y 431.934,Z 871.454,A -85,B 0,C 180,E1 20094.532,E2 20094.532} C_VEL
LIN {X 0,Y 430.5,Z 888.931,A -85,B 0,C 180,E1 20093.255,E2 20093.255} C_VEL
LIN {X 0,Y 429.117,Z 904.776,A -85,B 0,C 180,E1 20091.817,E2 20091.817} C_VEL
LIN {X 0,Y 427.833,Z 919.715,A -85,B 0,C 180,E1 20090.164,E2 20090.164} C_VEL
LIN {X 0,Y 426.653,Z 933.644,A -85,B 0,C 180,E1 20088.302,E2 20088.302} C_VEL
LIN {X 0,Y 425.691,Z 946.432,A -85,B 0,C 180,E1 20086.231,E2 20086.231} C_VEL
LIN {X 0,Y 424.997,Z 957.545,A -85,B 0,C 180,E1 20084.024,E2 20084.024} C_VEL
LIN {X 0,Y 424.592,Z 966.585,A -85,B 0,C 180,E1 20081.823,E2 20081.823} C_VEL
LIN {X 0,Y 424.416,Z 974.203,A -85,B 0,C 180,E1 20079.493,E2 20079.493} C_VEL
LIN {X 0,Y 424.388,Z 980.002,A -85,B 0,C 180,E1 20077.174,E2 20077.174} C_VEL
LIN {X 0,Y 424.46,Z 984.14,A -85,B 0,C 180,E1 20074.851,E2 20074.851} C_VEL
LIN {X 0,Y 424.552,Z 986.713,A -85,B 0,C 180,E1 20072.431,E2 20072.431} C_VEL
LIN {X 0,Y 424.605,Z 987.559,A -85,B 0,C 180,E1 20070.002,E2 20070.002} C_VEL
LIN {X 0,Y 424.56,Z 986.664,A -85,B 0,C 180,E1 20067.572,E2 20067.572} C_VEL
LIN {X 0,Y 424.471,Z 984.021,A -85,B 0,C 180,E1 20065.133,E2 20065.133} C_VEL
LIN {X 0,Y 424.4,Z 979.569,A -85,B 0,C 180,E1 20062.679,E2 20062.679} C_VEL
LIN {X 0,Y 424.436,Z 973.268,A -85,B 0,C 180,E1 20060.237,E2 20060.237} C_VEL
LIN {X 0,Y 424.637,Z 965.382,A -85,B 0,C 180,E1 20057.906,E2 20057.906} C_VEL
LIN {X 0,Y 425.106,Z 955.406,A -85,B 0,C 180,E1 20055.566,E2 20055.566} C_VEL
LIN {X 0,Y 425.85,Z 943.845,A -85,B 0,C 180,E1 20053.358,E2 20053.358} C_VEL
LIN {X 0,Y 426.882,Z 930.656,A -85,B 0,C 180,E1 20051.287,E2 20051.287} C_VEL
LIN {X 0,Y 428.127,Z 916.364,A -85,B 0,C 180,E1 20049.433,E2 20049.433} C_VEL
LIN {X 0,Y 429.493,Z 900.885,A -85,B 0,C 180,E1 20047.775,E2 20047.775} C_VEL
LIN {X 0,Y 430.976,Z 884.443,A -85,B 0,C 180,E1 20046.341,E2 20046.341} C_VEL
LIN {X 0,Y 432.412,Z 866.907,A -85,B 0,C 180,E1 20045.117,E2 20045.117} C_VEL
LIN {X 0,Y 433.716,Z 848.97,A -85,B 0,C 180,E1 20044.154,E2 20044.154} C_VEL
LIN {X 0,Y 434.815,Z 830.473,A -85,B 0,C 180,E1 20043.428,E2 20043.428} C_VEL
LIN {X 0,Y 435.573,Z 811.777,A -85,B 0,C 180,E1 20042.944,E2 20042.944} C_VEL
LIN {X 0,Y 438.104,Z 637.086,A -85,B 0,C 180,E1 20040.009,E2 20040.009} C_VEL
LIN {X 0,Y 435.751,Z 616.641,A -85,B 0,C 180,E1 20039.444,E2 20039.444} C_VEL
LIN {X 0,Y 439.897,Z 574.159,A -85,B 0,C 180,E1 20035.334,E2 20035.334} C_VEL
LIN {X 0,Y 440.552,Z 567.956,A -85,B 0,C 180,E1 20034.723,E2 20034.723} C_VEL
LIN {X 0,Y 434.938,Z 550.895,A -85,B 0,C 180,E1 20032.261,E2 20032.261} C_VEL
LIN {X 0,Y 429.243,Z 535.843,A -85,B 0,C 180,E1 20029.82,E2 20029.82} C_VEL
LIN {X 0,Y 425.333,Z 526.011,A -85,B 0,C 180,E1 20028.028,E2 20028.028} C_VEL
LIN {X 0,Y 425.317,Z 525.812,A -85,B 0,C 180,E1 20024.283,E2 20024.283} C_VEL
LIN {X 0,Y 425.315,Z 525.82,A -85,B 0,C 180,E1 20020.396,E2 20020.396} C_VEL
LIN {X 0,Y 425.279,Z 525.823,A -85,B 0,C 180,E1 20016.667,E2 20016.667} C_VEL
LIN {X 0,Y 425.264,Z 525.821,A -85,B 0,C 180,E1 20012.896,E2 20012.896} C_VEL
LIN {X 0,Y 425.262,Z 525.819,A -85,B 0,C 180,E1 20009.011,E2 20009.011} C_VEL
LIN {X 0,Y 425.277,Z 525.82,A -85,B 0,C 180,E1 20005.334,E2 20005.334} C_VEL
LIN {X 0,Y 425.301,Z 525.823,A -85,B 0,C 180,E1 20001.515,E2 20001.515} C_VEL
LIN {X 0,Y 425.294,Z 525.815,A -85,B 0,C 180,E1 19997.654,E2 19997.654} C_VEL
LIN {X 0,Y 425.262,Z 525.806,A -85,B 0,C 180,E1 19993.876,E2 19993.876} C_VEL
LIN {X 0,Y 425.239,Z 525.814,A -85,B 0,C 180,E1 19990.157,E2 19990.157} C_VEL
LIN {X 0,Y 425.242,Z 525.824,A -85,B 0,C 180,E1 19986.344,E2 19986.344} C_VEL
LIN {X 0,Y 425.26,Z 525.824,A -85,B 0,C 180,E1 19982.56,E2 19982.56} C_VEL
LIN {X 0,Y 425.3,Z 525.807,A -85,B 0,C 180,E1 19978.922,E2 19978.922} C_VEL
LIN {X 0,Y 425.302,Z 525.805,A -85,B 0,C 180,E1 19975.01,E2 19975.01} C_VEL
LIN {X 0,Y 425.276,Z 525.814,A -85,B 0,C 180,E1 19971.346,E2 19971.346} C_VEL
LIN {X 0,Y 425.266,Z 525.823,A -85,B 0,C 180,E1 19967.646,E2 19967.646} C_VEL
LIN {X 0,Y 425.27,Z 525.822,A -85,B 0,C 180,E1 19963.752,E2 19963.752} C_VEL
LIN {X 0,Y 425.293,Z 525.818,A -85,B 0,C 180,E1 19960.068,E2 19960.068} C_VEL
LIN {X 0,Y 425.318,Z 525.81,A -85,B 0,C 180,E1 19956.297,E2 19956.297} C_VEL
LIN {X 0,Y 425.323,Z 525.812,A -85,B 0,C 180,E1 19952.394,E2 19952.394} C_VEL
LIN {X 0,Y 425.311,Z 525.816,A -85,B 0,C 180,E1 19948.54,E2 19948.54} C_VEL
LIN {X 0,Y 425.333,Z 526.117,A -85,B 0,C 180,E1 19947.47,E2 19947.47} C_VEL
LIN {X 0,Y 430.143,Z 540.244,A -85,B 0,C 180,E1 19944.436,E2 19944.436} C_VEL
LIN {X 0,Y 434.422,Z 554.851,A -85,B 0,C 180,E1 19941.579,E2 19941.579} C_VEL
LIN {X 0,Y 436.207,Z 562.705,A -85,B 0,C 180,E1 19940.155,E2 19940.155} C_VEL
LIN {X 0,Y 433.51,Z 590.398,A -85,B 0,C 180,E1 19936.11,E2 19936.11} C_VEL
LIN {X 0,Y 431.114,Z 619.15,A -85,B 0,C 180,E1 19931.991,E2 19931.991} C_VEL
LIN {X 0,Y 430.292,Z 630.405,A -85,B 0,C 180,E1 19930.408,E2 19930.408} C_VEL
LIN {X 0,Y 431.692,Z 637.891,A -85,B 0,C 180,E1 19930.12,E2 19930.12} C_VEL
LIN {X 0,Y 434.607,Z 654.68,A -85,B 0,C 180,E1 19929.608,E2 19929.608} C_VEL
LIN {X 0,Y 432.769,Z 752.646,A -85,B 0,C 180,E1 19927.826,E2 19927.826} C_VEL
LIN {X 0,Y 432.292,Z 768.923,A -85,B 0,C 180,E1 19927.267,E2 19927.267} C_VEL
LIN {X 0,Y 431.606,Z 783.08,A -85,B 0,C 180,E1 19926.533,E2 19926.533} C_VEL
LIN {X 0,Y 430.713,Z 797.062,A -85,B 0,C 180,E1 19925.551,E2 19925.551} C_VEL
LIN {X 0,Y 429.612,Z 810.642,A -85,B 0,C 180,E1 19924.288,E2 19924.288} C_VEL
LIN {X 0,Y 428.612,Z 822.071,A -85,B 0,C 180,E1 19922.92,E2 19922.92} C_VEL
LIN {X 0,Y 427.581,Z 832.924,A -85,B 0,C 180,E1 19921.269,E2 19921.269} C_VEL
LIN {X 0,Y 426.679,Z 842,A -85,B 0,C 180,E1 19919.474,E2 19919.474} C_VEL
LIN {X 0,Y 426.015,Z 848.945,A -85,B 0,C 180,E1 19917.687,E2 19917.687} C_VEL
LIN {X 0,Y 425.738,Z 851.957,A -85,B 0,C 180,E1 19916.712,E2 19916.712} C_VEL
LIN {X 0,Y 424.536,Z 854.699,A -85,B 0,C 180,E1 19915.745,E2 19915.745} C_VEL
LIN {X 0,Y 420.028,Z 858.823,A -85,B 0,C 180,E1 19914.036,E2 19914.036} C_VEL
LIN {X 0,Y 417.454,Z 860.856,A -85,B 0,C 180,E1 19912.737,E2 19912.737} C_VEL
LIN {X 0,Y 417.131,Z 861.348,A -85,B 0,C 180,E1 19912.209,E2 19912.209} C_VEL
LIN {X 0,Y 417.033,Z 862.157,A -85,B 0,C 180,E1 19909.974,E2 19909.974} C_VEL
LIN {X 0,Y 417.072,Z 860.987,A -85,B 0,C 180,E1 19907.722,E2 19907.722} C_VEL
LIN {X 0,Y 417.242,Z 858.252,A -85,B 0,C 180,E1 19905.708,E2 19905.708} C_VEL
LIN {X 0,Y 417.592,Z 853.456,A -85,B 0,C 180,E1 19903.563,E2 19903.563} C_VEL
LIN {X 0,Y 418.104,Z 847.031,A -85,B 0,C 180,E1 19901.586,E2 19901.586} C_VEL
LIN {X 0,Y 418.807,Z 839.134,A -85,B 0,C 180,E1 19899.756,E2 19899.756} C_VEL
LIN {X 0,Y 419.652,Z 829.784,A -85,B 0,C 180,E1 19898.079,E2 19898.079} C_VEL
LIN {X 0,Y 420.599,Z 818.965,A -85,B 0,C 180,E1 19896.55,E2 19896.55} C_VEL
LIN {X 0,Y 421.596,Z 806.573,A -85,B 0,C 180,E1 19895.168,E2 19895.168} C_VEL
LIN {X 0,Y 422.566,Z 792.93,A -85,B 0,C 180,E1 19894.001,E2 19894.001} C_VEL
LIN {X 0,Y 423.347,Z 779.291,A -85,B 0,C 180,E1 19893.112,E2 19893.112} C_VEL
LIN {X 0,Y 424.004,Z 763.471,A -85,B 0,C 180,E1 19892.376,E2 19892.376} C_VEL
LIN {X 0,Y 424.37,Z 747.044,A -85,B 0,C 180,E1 19891.91,E2 19891.91} C_VEL
LIN {X 0,Y 425.731,Z 652.922,A -85,B 0,C 180,E1 19890.23,E2 19890.23} C_VEL
LIN {X 0,Y 421.858,Z 631.056,A -85,B 0,C 180,E1 19889.591,E2 19889.591} C_VEL
LIN {X 0,Y 422.003,Z 626.693,A -85,B 0,C 180,E1 19889.041,E2 19889.041} C_VEL
LIN {X 0,Y 424.191,Z 597.219,A -85,B 0,C 180,E1 19884.86,E2 19884.86} C_VEL
LIN {X 0,Y 426.475,Z 570.053,A -85,B 0,C 180,E1 19880.962,E2 19880.962} C_VEL
LIN {X 0,Y 427.201,Z 561.703,A -85,B 0,C 180,E1 19879.753,E2 19879.753} C_VEL
LIN {X 0,Y 422.431,Z 543.876,A -85,B 0,C 180,E1 19876.587,E2 19876.587} C_VEL
LIN {X 0,Y 417.373,Z 526.933,A -85,B 0,C 180,E1 19873.352,E2 19873.352} C_VEL
LIN {X 0,Y 417.355,Z 526.81,A -85,B 0,C 180,E1 19869.38,E2 19869.38} C_VEL
LIN {X 0,Y 417.323,Z 526.776,A -85,B 0,C 180,E1 19865.567,E2 19865.567} C_VEL
LIN {X 0,Y 417.304,Z 526.803,A -85,B 0,C 180,E1 19861.836,E2 19861.836} C_VEL
LIN {X 0,Y 417.295,Z 526.781,A -85,B 0,C 180,E1 19858.017,E2 19858.017} C_VEL
LIN {X 0,Y 417.311,Z 526.81,A -85,B 0,C 180,E1 19854.226,E2 19854.226} C_VEL
LIN {X 0,Y 417.343,Z 526.814,A -85,B 0,C 180,E1 19850.484,E2 19850.484} C_VEL
LIN {X 0,Y 417.347,Z 526.794,A -85,B 0,C 180,E1 19846.745,E2 19846.745} C_VEL
LIN {X 0,Y 417.319,Z 526.812,A -85,B 0,C 180,E1 19843.053,E2 19843.053} C_VEL
LIN {X 0,Y 417.308,Z 526.807,A -85,B 0,C 180,E1 19839.298,E2 19839.298} C_VEL
LIN {X 0,Y 417.313,Z 526.801,A -85,B 0,C 180,E1 19835.438,E2 19835.438} C_VEL
LIN {X 0,Y 417.331,Z 526.81,A -85,B 0,C 180,E1 19831.648,E2 19831.648} C_VEL
LIN {X 0,Y 417.363,Z 526.793,A -85,B 0,C 180,E1 19827.878,E2 19827.878} C_VEL
LIN {X 0,Y 417.368,Z 526.797,A -85,B 0,C 180,E1 19823.883,E2 19823.883} C_VEL
LIN {X 0,Y 417.348,Z 526.803,A -85,B 0,C 180,E1 19820.102,E2 19820.102} C_VEL
LIN {X 0,Y 417.32,Z 526.789,A -85,B 0,C 180,E1 19816.423,E2 19816.423} C_VEL
LIN {X 0,Y 417.321,Z 526.81,A -85,B 0,C 180,E1 19812.593,E2 19812.593} C_VEL
LIN {X 0,Y 417.329,Z 526.778,A -85,B 0,C 180,E1 19808.821,E2 19808.821} C_VEL
LIN {X 0,Y 417.362,Z 526.808,A -85,B 0,C 180,E1 19805.086,E2 19805.086} C_VEL
LIN {X 0,Y 417.373,Z 526.778,A -85,B 0,C 180,E1 19801.236,E2 19801.236} C_VEL
LIN {X 0,Y 417.36,Z 526.805,A -85,B 0,C 180,E1 19797.36,E2 19797.36} C_VEL
LIN {X 0,Y 417.34,Z 526.794,A -85,B 0,C 180,E1 19793.535,E2 19793.535} C_VEL
LIN {X 0,Y 417.332,Z 526.807,A -85,B 0,C 180,E1 19789.788,E2 19789.788} C_VEL
LIN {X 0,Y 417.333,Z 526.795,A -85,B 0,C 180,E1 19785.855,E2 19785.855} C_VEL
LIN {X 0,Y 417.355,Z 526.809,A -85,B 0,C 180,E1 19782.143,E2 19782.143} C_VEL
LIN {X 0,Y 417.384,Z 526.791,A -85,B 0,C 180,E1 19778.344,E2 19778.344} C_VEL
LIN {X 0,Y 417.377,Z 526.796,A -85,B 0,C 180,E1 19774.456,E2 19774.456} C_VEL
LIN {X 0,Y 417.37,Z 526.81,A -85,B 0,C 180,E1 19770.587,E2 19770.587} C_VEL
LIN {X 0,Y 417.353,Z 526.81,A -85,B 0,C 180,E1 19766.727,E2 19766.727} C_VEL
LIN {X 0,Y 417.345,Z 526.811,A -85,B 0,C 180,E1 19762.863,E2 19762.863} C_VEL
LIN {X 0,Y 417.347,Z 526.811,A -85,B 0,C 180,E1 19758.972,E2 19758.972} C_VEL
LIN {X 0,Y 417.356,Z 526.802,A -85,B 0,C 180,E1 19755.161,E2 19755.161} C_VEL
LIN {X 0,Y 417.413,Z 527.022,A -85,B 0,C 180,E1 19751.407,E2 19751.407} C_VEL
LIN {X 0,Y 425.034,Z 548.238,A -85,B 0,C 180,E1 19748.214,E2 19748.214} C_VEL
LIN {X 0,Y 432.166,Z 569.421,A -85,B 0,C 180,E1 19745.337,E2 19745.337} C_VEL
LIN {X 0,Y 427.89,Z 615.059,A -85,B 0,C 180,E1 19740.935,E2 19740.935} C_VEL
LIN {X 0,Y 427.87,Z 617.83,A -85,B 0,C 180,E1 19740.752,E2 19740.752} C_VEL
LIN {X 0,Y 430.387,Z 641.001,A -85,B 0,C 180,E1 19740.188,E2 19740.188} C_VEL
LIN {X 0,Y 427.683,Z 816.249,A -85,B 0,C 180,E1 19737.243,E2 19737.243} C_VEL
LIN {X 0,Y 426.8,Z 834.987,A -85,B 0,C 180,E1 19736.692,E2 19736.692} C_VEL
LIN {X 0,Y 425.636,Z 853.15,A -85,B 0,C 180,E1 19735.908,E2 19735.908} C_VEL
LIN {X 0,Y 424.291,Z 870.984,A -85,B 0,C 180,E1 19734.87,E2 19734.87} C_VEL
LIN {X 0,Y 422.854,Z 887.709,A -85,B 0,C 180,E1 19733.627,E2 19733.627} C_VEL
LIN {X 0,Y 421.388,Z 903.604,A -85,B 0,C 180,E1 19732.165,E2 19732.165} C_VEL
LIN {X 0,Y 420.035,Z 918.577,A -85,B 0,C 180,E1 19730.482,E2 19730.482} C_VEL
LIN {X 0,Y 418.795,Z 932.499,A -85,B 0,C 180,E1 19728.59,E2 19728.59} C_VEL
LIN {X 0,Y 417.803,Z 944.941,A -85,B 0,C 180,E1 19726.546,E2 19726.546} C_VEL
LIN {X 0,Y 417.067,Z 956.174,A -85,B 0,C 180,E1 19724.296,E2 19724.296} C_VEL
LIN {X 0,Y 416.635,Z 965.286,A -85,B 0,C 180,E1 19722.052,E2 19722.052} C_VEL
LIN {X 0,Y 416.451,Z 972.952,A -85,B 0,C 180,E1 19719.676,E2 19719.676} C_VEL
LIN {X 0,Y 416.436,Z 978.782,A -85,B 0,C 180,E1 19717.312,E2 19717.312} C_VEL
LIN {X 0,Y 416.524,Z 982.92,A -85,B 0,C 180,E1 19714.959,E2 19714.959} C_VEL
LIN {X 0,Y 416.633,Z 985.527,A -85,B 0,C 180,E1 19712.477,E2 19712.477} C_VEL
LIN {X 0,Y 416.692,Z 986.379,A -85,B 0,C 180,E1 19710.002,E2 19710.002} C_VEL
LIN {X 0,Y 416.639,Z 985.48,A -85,B 0,C 180,E1 19707.526,E2 19707.526} C_VEL
LIN {X 0,Y 416.535,Z 982.831,A -85,B 0,C 180,E1 19705.045,E2 19705.045} C_VEL
LIN {X 0,Y 416.446,Z 978.382,A -85,B 0,C 180,E1 19702.553,E2 19702.553} C_VEL
LIN {X 0,Y 416.473,Z 972.022,A -85,B 0,C 180,E1 19700.049,E2 19700.049} C_VEL
LIN {X 0,Y 416.68,Z 964.122,A -85,B 0,C 180,E1 19697.672,E2 19697.672} C_VEL
LIN {X 0,Y 417.139,Z 954.807,A -85,B 0,C 180,E1 19695.426,E2 19695.426} C_VEL
LIN {X 0,Y 417.914,Z 943.345,A -85,B 0,C 180,E1 19693.176,E2 19693.176} C_VEL
LIN {X 0,Y 418.956,Z 930.752,A -85,B 0,C 180,E1 19691.136,E2 19691.136} C_VEL
LIN {X 0,Y 420.268,Z 916.492,A -85,B 0,C 180,E1 19689.225,E2 19689.225} C_VEL
LIN {X 0,Y 421.741,Z 900.77,A -85,B 0,C 180,E1 19687.492,E2 19687.492} C_VEL
LIN {X 0,Y 423.299,Z 884.538,A -85,B 0,C 180,E1 19686.033,E2 19686.033} C_VEL
LIN {X 0,Y 424.808,Z 867.335,A -85,B 0,C 180,E1 19684.789,E2 19684.789} C_VEL
LIN {X 0,Y 426.152,Z 850.309,A -85,B 0,C 180,E1 19683.831,E2 19683.831} C_VEL
LIN {X 0,Y 427.367,Z 831.68,A -85,B 0,C 180,E1 19683.054,E2 19683.054} C_VEL
LIN {X 0,Y 428.227,Z 812.593,A -85,B 0,C 180,E1 19682.532,E2 19682.532} C_VEL
LIN {X 0,Y 430.949,Z 638.103,A -85,B 0,C 180,E1 19679.55,E2 19679.55} C_VEL
LIN {X 0,Y 428.526,Z 616.748,A -85,B 0,C 180,E1 19678.943,E2 19678.943} C_VEL
LIN {X 0,Y 433.202,Z 572.488,A -85,B 0,C 180,E1 19674.562,E2 19674.562} C_VEL
LIN {X 0,Y 433.269,Z 570.311,A -85,B 0,C 180,E1 19674.322,E2 19674.322} C_VEL
LIN {X 0,Y 427.809,Z 553.748,A -85,B 0,C 180,E1 19671.855,E2 19671.855} C_VEL
LIN {X 0,Y 421.608,Z 537.445,A -85,B 0,C 180,E1 19669.121,E2 19669.121} C_VEL
LIN {X 0,Y 417.369,Z 526.999,A -85,B 0,C 180,E1 19667.118,E2 19667.118} C_VEL
LIN {X 0,Y 417.338,Z 526.815,A -85,B 0,C 180,E1 19663.251,E2 19663.251} C_VEL
LIN {X 0,Y 417.335,Z 526.804,A -85,B 0,C 180,E1 19659.412,E2 19659.412} C_VEL
LIN {X 0,Y 417.354,Z 526.799,A -85,B 0,C 180,E1 19655.704,E2 19655.704} C_VEL
LIN {X 0,Y 417.373,Z 526.795,A -85,B 0,C 180,E1 19651.967,E2 19651.967} C_VEL
LIN {X 0,Y 417.337,Z 526.799,A -85,B 0,C 180,E1 19648.318,E2 19648.318} C_VEL
LIN {X 0,Y 417.316,Z 526.807,A -85,B 0,C 180,E1 19644.638,E2 19644.638} C_VEL
LIN {X 0,Y 417.313,Z 526.812,A -85,B 0,C 180,E1 19640.769,E2 19640.769} C_VEL
LIN {X 0,Y 417.321,Z 526.815,A -85,B 0,C 180,E1 19636.995,E2 19636.995} C_VEL
LIN {X 0,Y 417.348,Z 526.799,A -85,B 0,C 180,E1 19633.296,E2 19633.296} C_VEL
LIN {X 0,Y 417.348,Z 526.793,A -85,B 0,C 180,E1 19629.376,E2 19629.376} C_VEL
LIN {X 0,Y 417.317,Z 526.806,A -85,B 0,C 180,E1 19625.775,E2 19625.775} C_VEL
LIN {X 0,Y 417.309,Z 526.814,A -85,B 0,C 180,E1 19622.059,E2 19622.059} C_VEL
LIN {X 0,Y 417.317,Z 526.811,A -85,B 0,C 180,E1 19618.215,E2 19618.215} C_VEL
LIN {X 0,Y 417.339,Z 526.798,A -85,B 0,C 180,E1 19614.501,E2 19614.501} C_VEL
LIN {X 0,Y 417.37,Z 526.793,A -85,B 0,C 180,E1 19610.763,E2 19610.763} C_VEL
LIN {X 0,Y 417.372,Z 526.795,A -85,B 0,C 180,E1 19606.845,E2 19606.845} C_VEL
LIN {X 0,Y 417.346,Z 526.802,A -85,B 0,C 180,E1 19603.148,E2 19603.148} C_VEL
LIN {X 0,Y 417.337,Z 526.803,A -85,B 0,C 180,E1 19599.379,E2 19599.379} C_VEL
LIN {X 0,Y 417.339,Z 526.802,A -85,B 0,C 180,E1 19595.513,E2 19595.513} C_VEL
LIN {X 0,Y 417.353,Z 526.812,A -85,B 0,C 180,E1 19591.682,E2 19591.682} C_VEL
LIN {X 0,Y 417.423,Z 527.084,A -85,B 0,C 180,E1 19588.338,E2 19588.338} C_VEL
LIN {X 0,Y 422.477,Z 541.82,A -85,B 0,C 180,E1 19585.059,E2 19585.059} C_VEL
LIN {X 0,Y 426.562,Z 555.574,A -85,B 0,C 180,E1 19582.281,E2 19582.281} C_VEL
LIN {X 0,Y 428.903,Z 565.714,A -85,B 0,C 180,E1 19580.387,E2 19580.387} C_VEL
LIN {X 0,Y 426.047,Z 593.435,A -85,B 0,C 180,E1 19576.28,E2 19576.28} C_VEL
LIN {X 0,Y 423.546,Z 621.742,A -85,B 0,C 180,E1 19572.161,E2 19572.161} C_VEL
LIN {X 0,Y 422.897,Z 630.387,A -85,B 0,C 180,E1 19570.939,E2 19570.939} C_VEL
LIN {X 0,Y 424.065,Z 636.631,A -85,B 0,C 180,E1 19570.683,E2 19570.683} C_VEL
LIN {X 0,Y 427.461,Z 655.689,A -85,B 0,C 180,E1 19570.076,E2 19570.076} C_VEL
LIN {X 0,Y 425.51,Z 753.242,A -85,B 0,C 180,E1 19568.268,E2 19568.268} C_VEL
LIN {X 0,Y 425.004,Z 769.436,A -85,B 0,C 180,E1 19567.705,E2 19567.705} C_VEL
LIN {X 0,Y 424.255,Z 784.087,A -85,B 0,C 180,E1 19566.933,E2 19566.933} C_VEL
LIN {X 0,Y 423.306,Z 798.033,A -85,B 0,C 180,E1 19565.936,E2 19565.936} C_VEL
LIN {X 0,Y 422.205,Z 810.787,A -85,B 0,C 180,E1 19564.738,E2 19564.738} C_VEL
LIN {X 0,Y 421.175,Z 821.935,A -85,B 0,C 180,E1 19563.414,E2 19563.414} C_VEL
LIN {X 0,Y 420.037,Z 833.006,A -85,B 0,C 180,E1 19561.735,E2 19561.735} C_VEL
LIN {X 0,Y 419.086,Z 841.936,A -85,B 0,C 180,E1 19559.996,E2 19559.996} C_VEL
LIN {X 0,Y 418.295,Z 849.48,A -85,B 0,C 180,E1 19558.088,E2 19558.088} C_VEL
LIN {X 0,Y 417.69,Z 855.504,A -85,B 0,C 180,E1 19555.976,E2 19555.976} C_VEL
LIN {X 0,Y 417.334,Z 859.274,A -85,B 0,C 180,E1 19554.031,E2 19554.031} C_VEL
LIN {X 0,Y 417.131,Z 861.348,A -85,B 0,C 180,E1 19552.209,E2 19552.209} C_VEL
LIN {X 0,Y 416.072,Z 862.122,A -85,B 0,C 180,E1 19551.154,E2 19551.154} C_VEL
LIN {X 0,Y 411.808,Z 862.846,A -85,B 0,C 180,E1 19549.31,E2 19549.31} C_VEL
LIN {X 0,Y 409.422,Z 862.387,A -85,B 0,C 180,E1 19547.949,E2 19547.949} C_VEL
LIN {X 0,Y 409.177,Z 861.878,A -85,B 0,C 180,E1 19547.409,E2 19547.409} C_VEL
LIN {X 0,Y 409.408,Z 858.502,A -85,B 0,C 180,E1 19545.145,E2 19545.145} C_VEL
LIN {X 0,Y 409.789,Z 853.638,A -85,B 0,C 180,E1 19543.113,E2 19543.113} C_VEL
LIN {X 0,Y 410.386,Z 846.913,A -85,B 0,C 180,E1 19541.095,E2 19541.095} C_VEL
LIN {X 0,Y 411.2,Z 838.287,A -85,B 0,C 180,E1 19539.169,E2 19539.169} C_VEL
LIN {X 0,Y 412.097,Z 828.85,A -85,B 0,C 180,E1 19537.526,E2 19537.526} C_VEL
LIN {X 0,Y 413.159,Z 817.241,A -85,B 0,C 180,E1 19535.933,E2 19535.933} C_VEL
LIN {X 0,Y 414.21,Z 804.414,A -85,B 0,C 180,E1 19534.567,E2 19534.567} C_VEL
LIN {X 0,Y 415.19,Z 790.857,A -85,B 0,C 180,E1 19533.45,E2 19533.45} C_VEL
LIN {X 0,Y 416.05,Z 775.582,A -85,B 0,C 180,E1 19532.512,E2 19532.512} C_VEL
LIN {X 0,Y 416.656,Z 759.387,A -85,B 0,C 180,E1 19531.837,E2 19531.837} C_VEL
LIN {X 0,Y 416.973,Z 742.714,A -85,B 0,C 180,E1 19531.43,E2 19531.43} C_VEL
LIN {X 0,Y 418.347,Z 653.991,A -85,B 0,C 180,E1 19529.823,E2 19529.823} C_VEL
LIN {X 0,Y 414.226,Z 630.386,A -85,B 0,C 180,E1 19529.099,E2 19529.099} C_VEL
LIN {X 0,Y 416.452,Z 601.041,A -85,B 0,C 180,E1 19524.902,E2 19524.902} C_VEL
LIN {X 0,Y 418.825,Z 573.733,A -85,B 0,C 180,E1 19520.934,E2 19520.934} C_VEL
LIN {X 0,Y 419.654,Z 563.977,A -85,B 0,C 180,E1 19519.497,E2 19519.497} C_VEL
LIN {X 0,Y 414.977,Z 546.505,A -85,B 0,C 180,E1 19516.342,E2 19516.342} C_VEL
LIN {X 0,Y 410.22,Z 530.523,A -85,B 0,C 180,E1 19513.285,E2 19513.285} C_VEL
LIN {X 0,Y 409.386,Z 527.898,A -85,B 0,C 180,E1 19512.7,E2 19512.7} C_VEL
LIN {X 0,Y 409.392,Z 527.803,A -85,B 0,C 180,E1 19508.902,E2 19508.902} C_VEL
LIN {X 0,Y 409.408,Z 527.766,A -85,B 0,C 180,E1 19505.162,E2 19505.162} C_VEL
LIN {X 0,Y 409.4,Z 527.771,A -85,B 0,C 180,E1 19501.256,E2 19501.256} C_VEL
LIN {X 0,Y 409.369,Z 527.779,A -85,B 0,C 180,E1 19497.499,E2 19497.499} C_VEL
LIN {X 0,Y 409.362,Z 527.798,A -85,B 0,C 180,E1 19493.709,E2 19493.709} C_VEL
LIN {X 0,Y 409.366,Z 527.803,A -85,B 0,C 180,E1 19489.851,E2 19489.851} C_VEL
LIN {X 0,Y 409.385,Z 527.794,A -85,B 0,C 180,E1 19486.085,E2 19486.085} C_VEL
LIN {X 0,Y 409.409,Z 527.782,A -85,B 0,C 180,E1 19482.273,E2 19482.273} C_VEL
